FUNCTION_BLOCK TFPalletizerWorkAreaManagerTF_Lastre
VAR_INPUT
	Cfg 						: Config;
	WorkArea 					: POINTER TO ARRAY [1..MAXAREA] OF TFMachinePalletizer_WorkArea;
	WorkAreaState 				: POINTER TO ARRAY [1..MAXAREA] OF TFMachinePalletizer_WorkAreaState;
	WorkAreaOffset				: POINTER TO ARRAY [1..MAXAREA] OF TFMachinePalletizer_WorkAreaOffset;
	PX_WorkArea 				: ARRAY [1..MAXAREA] OF BOOL;
	WorkPickPoint 				: POINTER TO ARRAY [1..MAXPICKPOINT] OF TFMachinePalletizer_WorkPickPointSlab;
	WorkPickPointState 			: POINTER TO ARRAY [1..MAXPICKPOINT] OF TFMachinePalletizer_WorkPickPoint_State;
	//WorkPickPointTransportState	: POINTER TO ARRAY [1..MAXPICKPOINT] OF TFMachinePalletizer_WorkPickPointTransport_State;
	//WorkPickPointStoreState		: POINTER TO ARRAY [1..MAXPICKPOINT] OF TFMachinePalletizer_WorkPickPointStore_State;
	WorkPickPointOffset 		: POINTER TO ARRAY [1..MAXPICKPOINT] OF TFMachinePalletizer_WorkPickPointOffset;
	Forming 					: POINTER TO ARRAY [1..MAXFORMING] OF TFMachinePalletizer_FormingForSlab;
	Pallet 						: POINTER TO ARRAY [1..MAXPALLET] OF TFMachinePalletizer_Pallet;
	Layer 						: POINTER TO ARRAY [1..MAXLAYER] OF TFMachinePalletizer_Layer;
	Mission 					: POINTER TO TFMachinePalletizer_Mission;
	PickPlaceParameters			: POINTER TO TFMachinePalletizer_PickPlaceParameters;
	ExternalWaitPositionRequest : BOOL;
	ProgressiveNrWA 			: POINTER TO UDINT;
	UsedCode 					: POINTER TO ARRAY [1..MAXFORMINGCODE] OF INT;
	TCPParameter 				: POINTER TO TFModulePalletizerRobot_TCPPar;
	TilterPack 					: POINTER TO ARRAY [1..MAXHANDLINGSTACK] OF TFHandlingPack;
	PreviousPWA 				: POINTER TO UINT;
	RestoreCWA 					: POINTER TO BOOL;
	PreviousStackWA 			: POINTER TO INT;
	WorkAreaManager 			: POINTER TO TFWorkAreaManager;
	ModuleAX_X 					: POINTER TO TFModulePalletizer_Ax;
	ModuleAX_Y 					: POINTER TO TFModulePalletizer_Ax;
	ModuleAX_Z 					: POINTER TO TFModulePalletizer_Ax;
	ModuleAX_J 					: POINTER TO TFModulePalletizer_Ax;
	ModuleAX_K 					: POINTER TO TFModulePalletizer_Ax;
	
	ModulePinza					: pointer to TFModulePalletizer_Pinza;
	
	WorkAreaZone 				: POINTER TO TFMachinePalletizer_WorkAreaZone;	// Struttura delle zone di lavoro
	//HandlingPackTable : POINTER TO TFHandlingPackTable;						// Tabella contenente i pacchi sui trasporti
	ArrayPacchi 			: POINTER TO DUT_ArrayPacchi; 						//Array contenente i pacchi sui trasporti				
	GestioneAZoneAbilitata 	: POINTER TO BOOL;									// Abilitazione della gestione a zone
	HandlingRun 			: BOOL;												//Traspoti in Automatico
	RichiestaStartRibaltino : BOOL;
	AbilitaForzaturaStatoDaRiposoAPrelievo 			: POINTER TO BOOL;			// Abilita il cambio al volo della missione dal ciclo di riposo al ciclo di prelievo
	AbilitaDisposizionePalletContinua 				: POINTER TO BOOL;			// Abilitazione del deposito dei pallet ogni qualvolta il carico imposto dalla line a soddisfi determinato requisiti
	AbilitaDepositoPaccoOrrizzonataleConTasteggio 	: POINTER TO BOOL; 			// Abilitazione per il deposito del pacco con tasteggio del pacco orrizzontale
	AbilitaAssegnazioneCodicePiazzoleConPaccoSuRibaltino 	: BOOL := TRUE; 	// Abilitazione della gestione del codice in modo opportunistico rispettando le zone
	AbilitaOffsetInUscitaTasteggioPrelievoPallet 			: POINTER TO BOOL; 	// Abilitazione dell'offset in uscita dei tastatori in prelievo pallet con tasteggio
	
	//TabellaDiProduzione : POINTER TO ARRAY [1..MAXPRODLIST] OF TFMachinePalletizer_ListaProduzione; //Lista degli ordini di produzione che devo Svolgere
	
	WorkAreaProductionList : POINTER TO ARRAY [1..MAXAREA] OF TFMachinePalletizer_ListaProduzione_WAM;// ARRAY [1..MAXAREA] OF TFMachinePalletizer_ListaProduzione_WAM; //Lista di produzione che devo Svolgere PER ogni POSTAZIONE
	
	//
	RichiestaIngZonaDX : BOOL; //Richiesta di ingresso zona DX del pallettizzatore, le postazioni vanno dalla 1 alla 4
	RichiestaIngZonaSX : BOOL; //Richiesta di ingresso zona SX del pallettizzatore, le postazioni vanno dalla 5 alla 8
	
END_VAR
VAR_OUTPUT
	InWaitPosition 			: BOOL;
	DepositoPaccoInLenta 	: BOOL;					// TRUE: Il deposito del pacco deve avvenire in lenta
	ForzaPrelievoPaccoDuranteCicloDiRiposo : BOOL; 	// Indica che il ciclo sta facendo un salto: Da ciclo di riposo -> A ciclo di prelievo 
	Errore : TFError_WAM; 							//Codice di errore del WorkAreaManager
END_VAR
VAR
	i : UINT;
	TimerPositionMission : REAL;
	CurrentWorkArea : INT;
	cwa : UINT;
	pwa : UINT;
	wa : INT;
	pf : INT;
	pp : INT;
	fcode : INT;
	ppick : UINT; //Punto di prelievo
	XPick : LREAL;
	YPick : LREAL;
	ZPick : LREAL;
	JPick : LREAL;
	EnableCode : ARRAY [1..MAXFORMINGCODE*MAXFORMING] OF INT;
	WAPointer : ARRAY [1..MAXAREA] OF TFMachinePalletizer_WorkAreaSort;
	ZOffsetPick : REAL;
	ZOffsetPlace : REAL;
	WaitPositionRequest : BOOL;
	WaitPositionRequestTRIG : BOOL;
	BypassTEST 								: BOOL; // ByPASS per il conteggio dei pacchi durante le simulazioni
	CicloDiRiposoNecessario 				: BOOL;	// Forzatura del ciclo di riposo da parte del WAManager
	NPacchiPresentiSuLinea 					: UINT;	// Indica il numero dei pacchi presenti sulla linea
	NUltimiTrasportiOccupati 				: UINT;	// Indica il numero di trasporti occupati a partire dal ribaltino
	HandlingOKPrelievoPacco 				: BOOL; // Indica che il Ribaltino è pronto a consegnare il pacco
	ConsentiDepositoPaccoSuWA 				: BOOL; // Indica il Pacco può essere depositato sulla WorkArea

	DisabilitaApproccioPacciOrrizzontali 	: BOOL := TRUE; // Abilitazione dell'approccio per i pacchi orrizzontali, in questo modo il ciclo è più rapido
	QuotaFittizziaPerTasteggioDepPacchi 	: REAL := 200; 	//Quota fittizzia per consentire il tasteggio durante il deposito dei pacci orrizzontali
	UltimaPoastazioneDiAssegnazione 		: INT;	// Variabile per Debug Interno
	UltimoComando 							: INT;	// Variabile per Debug Interno
	UltimoStatoCMDRibaltino 				: INT;	// Variabile per Debug Interno
	WAconCodiceWPPPresente 					: BOOL;	// Indica che esiste almento una WA in lavorazione con il codice del pacco presente sul ribaltino in questione
	FormaturaAttivaMista 					: BOOL;	// Indica che la formatura attiva è di tipo Misto (FALSE:utilizzata per anticipare ulteriormente il ribaltino,TRUE:si aspetta che sia terminato il deposito del pacco in corso prima di comandare il ribaltino)
	PalletDepositatiSenzaCodicePresenti 	: BOOL;	// Indica che sono presenti dei pallet depositati con codice 0 ( Per assegnazione codice in modalità opportunistica(In base al codice sul ribaltino))
	CodiceValidoPerWA 						: BOOL; // Indica che il codice del pacco sul ribaltino è presente nella formatura attiva nella WA considerata

	SimulazioneSenzaPallet 					: BOOL; //Variabile per simulare in officina senza pacco e pallet
	
	FormatureMultipleAttive 				: BOOL;	//Indica che ci sono più formature Diverse ABILITATE
	////////// NUOVE PER LASTRE ////////////
	DIREZIONE_X_POSITIVA					: BOOL;
	
	TFWAM_CreaMissione_DepFaldaSuLastra 	: TFWAM_CreaMissione_DepPrelElemento;
	TFWAM_CreaMissione_DepFaldaSuPallet 	: TFWAM_CreaMissione_DepPrelElemento;
	TFWAM_CreaMissione_Destinazione			: TFWAM_CreaMissione_DepPrelElemento;
	
	TFWAM_CreaMissione_PrelLastraDaWA 		: TFWAM_CreaMissione_DepPrelElemento;
	TFWAM_CreaMissione_DepLastraDaWA		: TFWAM_CreaMissione_DepPrelElemento;
	
	TFWAM_CreaMissione_DepLastraDaPP		: TFWAM_CreaMissione_DepPrelElemento;
	
	TFWAM_CreaMissione_DepFaldaSuMagazzino 	: TFWAM_CreaMissione_DepPrelElemento;

	
	PostazioneConListaInEsecuzione : UINT; //Indica il numero della postazione avente una lista di lavorazione ion esecuzione
	WADiDepositoFinale : UINT; //WorkArea Di Desinazione della Lastra 
	NLastraDaPrelevare : INT; //Numero della lastra da prelevare = N° della prima lastra che sarà prelevata dalla cavallina
	RIESEGUI_PAREGGIATURA : BOOL; //Forzo L'esecuzione della pareggiatura della lastra Dopo arresto anomalo del ciclo
	ElList1: UINT;
	ElList : UINT;//Elemento in elaborazione nella lista
	
	
	LastRequetsID : STRING; //Ultimo ID depositato sulla rulliera dopo il depal
	LatoPrelievo : INT; //Indica il lato di prelievo per le cavalline = 90 o 180
	LastPpick : UINT; //Memoria dell'ultimo 

	debug : bool;
	ppickOld : UINT;
	ApprendimentoNulloRullieraDeposito : TFMachinePalletizer_CoordinateApprendimento;
	DisabilitaCicloRiposoPerPezzoInPresa : BOOL;
	LatoDeposito : INT; //Indica il lato di deposito.. per le cavalline = 90 o 180


	Debug_SupportoMancanteInDeposito : BOOL;//Indica che il supporto sul deposito non è presente
	Debug_RullieraInManuale : BOOL;//Indica che la rulliera è in manuale
	Debug_NessunaListaDaProcessare : BOOL;//Indica che non c'è nessuna lista da processare
	Debug_RicSupportoWA : ARRAY[1..MAXAREA] OF BOOL;//Indica una richiesta del supporto da partede della postazione
	Actual_WorkOrde: INT;
	AltezzaCentroLastraInclinata : REAL;
	AngoloPrelievo : REAL;
	QuotaLastraYRealTimePrelievo : REAL;
	QuotaLastraYRealTimeDeposito : REAL;
	QuotaLastraZRealTimePrelievo : REAL;
	QuotaLastraZRealTimeDeposito : REAL;
	
	TFCalcoloFormaturaDaLista	: Calcolo_Formatura_Completa;//FB per il calcolo della formatura
	CalcolaFormaturaTrig : BOOL;
	
	PplaceOld : UINT;
	AngoloDepositoLastra : REAL;
	
	Y_PuntoPrelievo0: REAL;
	Y_PuntoPrelievo180: REAL;
	OffSetY180Cavallete: REAL;
	AguloDeRecogida: UINT;
	AguloDeDeposito: UINT;
END_VAR

(* Set variabili varie *)
Errore.Code:= 0;
Errore.Extracode:=0;

(* Chiamata del timer per andare alla posizione di riposo *)
TFTimerCall(ADR(TimerPositionMission),Cfg.TimeBase);
(* Inizializzazione del WAM *)
IF WorkAreaManager^.State = -1 THEN
	WorkAreaManager^.State := WAMANAGER_NOP;
	ExternalWaitPositionRequest := TRUE;
END_IF

EnableCode := TFGetEnableCode_Lastre(Forming);



IF Mission^.State <> MISSION_STATE_NOP THEN
	TFTimerSet(ADR(TimerPositionMission),300,TRUE);
END_IF
IF ((ExternalWaitPositionRequest AND WorkAreaManager^.State = WAMANAGER_NOP)  OR TFTimerDone(ADR(TimerPositionMission))) AND NOT InWaitPosition THEN
	CicloDiRiposoNecessario	:= TRUE;
	WaitPositionRequestTRIG := TRUE;
END_IF
IF 	WaitPositionRequestTRIG THEN
	WaitPositionRequest := TRUE;
END_IF
IF WaitPositionRequestTRIG AND WaitPositionRequest AND (InWaitPosition AND WorkAreaManager^.State = WAMANAGER_NOP) THEN
	WaitPositionRequest := FALSE;
	WaitPositionRequestTRIG := FALSE;
END_IF


CASE WorkAreaManager^.State OF
	WAMANAGER_NOP:
			
		IF RichiestaIngZonaSX THEN
			Mission^.PPick			:= 5;
			Mission^.TPick 			:= TPICK_NOT_DEFINED;
			Mission^.XPick			:= WorkArea^[5].X;
			Mission^.YPick			:= WorkSpace.Y/2 + OffSetPosYReposo;//Workarea^[5].Y;
			Mission^.ZPick			:= ModuleAX_Z^.Ax^.Parameter.MAXPosition - 100 -OffsetSicurezza.Z.Avuoto; // estaba 100
			
			Mission^.JPick			:= 90;
			
			Mission^.PPlace			:= Mission^.PPick;
			Mission^.XPlace			:= Mission^.XPick;
			Mission^.YPlace			:= Mission^.YPick;
			Mission^.ZPlace			:= Mission^.ZPick;
			Mission^.JPlace			:= Mission^.JPick;

			Mission^.XDim 	:= 0;
			Mission^.YDim	:= 0;
			Mission^.ZDim	:= 0;
			
			X_Riposo := Mission^.XPick;
			Y_Riposo := Mission^.YPick;
			Z_Riposo := Mission^.ZPick;
			J_Riposo := Mission^.JPick;
			
			(* Set della condizione di posizione di riposo Wait Position *)
			InWaitPosition := TFPalletizerInPosizioneRiposo(ModuleAX_X,ModuleAX_Y,ModuleAX_Z,ModuleAX_J,Mission);

			IF WaitPositionRequest AND NOT InWaitPosition AND
			(ExternalWaitPositionRequest OR CicloDiRiposoNecessario) THEN //Se la macchina non è a riposo, ce la mando
				WorkAreaManager^.State := WAMANAGER_CICLO_RIPOSO_INIT;
			ELSE	//Se la macchina è ferma e a riposo -> verifica eventuali cambi di produzione
				ReadyToChange := TRUE;
			END_IF

		ELSIF RichiestaIngZonaDX THEN
			Mission^.PPick			:= 1;
			Mission^.TPick 			:= TPICK_NOT_DEFINED;
			Mission^.XPick			:= WorkArea^[4].X;
			Mission^.YPick			:= WorkSpace.Y/2 + OffSetPosYReposo;//Workarea^[1].Y;
			Mission^.ZPick			:= ModuleAX_Z^.Ax^.Parameter.MAXPosition - 100 -OffsetSicurezza.Z.Avuoto ;
			Mission^.JPick			:= 90;
			
			Mission^.PPlace			:= Mission^.PPick;
			Mission^.XPlace			:= Mission^.XPick;
			Mission^.YPlace			:= Mission^.YPick;
			Mission^.ZPlace			:= Mission^.ZPick;
			Mission^.JPlace			:= Mission^.JPick;

			Mission^.XDim 	:= 0;
			Mission^.YDim	:= 0;
			Mission^.ZDim	:= 0;
			
			X_Riposo := Mission^.XPick;
			Y_Riposo := Mission^.YPick;
			Z_Riposo := Mission^.ZPick;
			J_Riposo := Mission^.JPick;

			(* Set della condizione di posizione di riposo Wait Position *)
			InWaitPosition := TFPalletizerInPosizioneRiposo(ModuleAX_X,ModuleAX_Y,ModuleAX_Z,ModuleAX_J,Mission);
			
			IF WaitPositionRequest AND NOT InWaitPosition AND
			(ExternalWaitPositionRequest OR CicloDiRiposoNecessario) THEN //Se la macchina non è a riposo, ce la mando
				WorkAreaManager^.State := WAMANAGER_CICLO_RIPOSO_INIT;
			ELSE	//Se la macchina è ferma e a riposo -> verifica eventuali cambi di produzione
				ReadyToChange := TRUE;
			END_IF
		ELSE
		 	Mission^.PPick			:= 1;
			Mission^.TPick 			:= TPICK_NOT_DEFINED;
			Mission^.XPick			:= ModuleAX_X^.Ax^.Status.ActPosition;// WorkArea^[1].X;
			Mission^.YPick			:= WorkSpace.Y/2 + OffSetPosYReposo;//Workarea^[1].Y;
			Mission^.ZPick			:= ModuleAX_Z^.Ax^.Parameter.MAXPosition - 100 - OffsetSicurezza.Z.Avuoto; 
			Mission^.JPick			:= 90;
			
			Mission^.PPlace			:= Mission^.PPick;
			Mission^.XPlace			:= Mission^.XPick;
			Mission^.YPlace			:= Mission^.YPick;
			Mission^.ZPlace			:= Mission^.ZPick;
			Mission^.JPlace			:= Mission^.JPick;

			Mission^.XDim 	:= 0;
			Mission^.YDim	:= 0;
			Mission^.ZDim	:= 0;
			
			X_Riposo := Mission^.XPick;
			Y_Riposo := Mission^.YPick;
			Z_Riposo := Mission^.ZPick;
			J_Riposo := Mission^.JPick;

			(* Set della condizione di posizione di riposo Wait Position *)
			InWaitPosition := TFPalletizerInPosizioneRiposo(ModuleAX_X,ModuleAX_Y,ModuleAX_Z,ModuleAX_J,Mission);
			
			IF WaitPositionRequest AND NOT InWaitPosition AND
			(ExternalWaitPositionRequest OR CicloDiRiposoNecessario) THEN //Se la macchina non è a riposo, ce la mando
				WorkAreaManager^.State := WAMANAGER_CICLO_RIPOSO_INIT;
			ELSE	//Se la macchina è ferma e a riposo -> verifica eventuali cambi di produzione
				ReadyToChange := TRUE;
			END_IF
		END_IF
						
	WAMANAGER_CICLO_RIPOSO_INIT:
	 	
		IF RichiestaIngZonaSX THEN
			Mission^.PPick			:= 5;
			Mission^.TPick 			:= TPICK_NOT_DEFINED;
			IF AreaPikingConCavallete AND MultiplesCavalletesReceta OR WorkAreaState^[PosRobot].Supporto.Tipologia = CAVALLETTO 
				OR (PosRobot <> 0 AND  HMI_WorkAreaDataPicking[PosRobot].Typology = CAVALLETTO)	THEN
				Mission^.XPick			:= WorkArea^[PosFinOrdenPikingCaballete].X;
				Mission^.YPick			:= ModuleAX_y^.Ax^.AxRef^.NcToPlc.ActPos;
				Mission^.ZPick			:= ModuleAX_Z^.Ax^.Parameter.MAXPosition - 100 -OffsetSicurezza.Z.Avuoto;
				Mission^.JPick			:= ModuleAX_j^.Ax^.AxRef^.NcToPlc.ActPos ;
			ELSE
				Mission^.XPick			:= WorkArea^[5].X;
				Mission^.YPick			:= WorkSpace.Y/2 + OffSetPosYReposo;//Workarea^[5].Y;
				Mission^.ZPick			:= ModuleAX_Z^.Ax^.Parameter.MAXPosition - 100 -OffsetSicurezza.Z.Avuoto;
				Mission^.JPick			:= 90;
			END_IF
			
			Mission^.PPlace			:= Mission^.PPick;
			Mission^.XPlace			:= Mission^.XPick;
			Mission^.YPlace			:= Mission^.YPick;
			Mission^.ZPlace			:= Mission^.ZPick;
			Mission^.JPlace			:= Mission^.JPick;

			Mission^.XDim 	:= 0;
			Mission^.YDim	:= 0;
			Mission^.ZDim	:= 0;
			
			X_Riposo := Mission^.XPick;
			Y_Riposo := Mission^.YPick;
			Z_Riposo := Mission^.ZPick;
			J_Riposo := Mission^.JPick;

		ELSIF RichiestaIngZonaDX THEN
			Mission^.PPick			:= 1;
			Mission^.TPick 			:= TPICK_NOT_DEFINED;
			IF AreaPikingConCavallete AND MultiplesCavalletesReceta OR WorkAreaState^[PosRobot].Supporto.Tipologia = CAVALLETTO 
				OR (PosRobot <> 0 AND  HMI_WorkAreaDataPicking[PosRobot].Typology = CAVALLETTO) THEN
				Mission^.XPick			:= WorkArea^[PosFinOrdenPikingCaballete].X;
				Mission^.YPick			:= ModuleAX_y^.Ax^.AxRef^.NcToPlc.ActPos;
				Mission^.ZPick			:= ModuleAX_Z^.Ax^.Parameter.MAXPosition - 100 -OffsetSicurezza.Z.Avuoto;
				Mission^.JPick			:= ModuleAX_j^.Ax^.AxRef^.NcToPlc.ActPos ;
				
				
			ELSE
				Mission^.XPick			:= WorkArea^[4].X;
				Mission^.YPick			:= WorkSpace.Y/2+OffSetPosYReposo;//Workarea^[1].Y;
				Mission^.ZPick			:= ModuleAX_Z^.Ax^.Parameter.MAXPosition - 100 -OffsetSicurezza.Z.Avuoto;
				Mission^.JPick			:= 90;
			END_IF
			
			
			Mission^.PPlace			:= Mission^.PPick;
			Mission^.XPlace			:= Mission^.XPick;
			Mission^.YPlace			:= Mission^.YPick;
			Mission^.ZPlace			:= Mission^.ZPick;
			Mission^.JPlace			:= Mission^.JPick;

			Mission^.XDim 	:= 0;
			Mission^.YDim	:= 0;
			Mission^.ZDim	:= 0;
			
			X_Riposo := Mission^.XPick;
			Y_Riposo := Mission^.YPick;
			Z_Riposo := Mission^.ZPick;
			J_Riposo := Mission^.JPick;
		ELSE
		 	Mission^.PPick			:= 1;
			Mission^.TPick 			:= TPICK_NOT_DEFINED;
			IF AreaPikingConCavallete AND MultiplesCavalletesReceta OR WorkAreaState^[PosRobot].Supporto.Tipologia = CAVALLETTO
				OR (PosRobot <> 0 AND  HMI_WorkAreaDataPicking[PosRobot].Typology = CAVALLETTO) THEN
				Mission^.XPick			:= WorkArea^[PosFinOrdenPikingCaballete].X;
				Mission^.YPick			:= ModuleAX_y^.Ax^.AxRef^.NcToPlc.ActPos;
				Mission^.ZPick			:= ModuleAX_Z^.Ax^.Parameter.MAXPosition - 100 -OffsetSicurezza.Z.Avuoto;
				Mission^.JPick			:= ModuleAX_j^.Ax^.AxRef^.NcToPlc.ActPos ;
			ELSE
				Mission^.XPick			:= ModuleAX_X^.Ax^.Status.ActPosition;// WorkArea^[1].X;
				Mission^.YPick			:= (*2000   *)   WorkSpace.Y/2+OffSetPosYReposo;//Workarea^[1].Y ;
				Mission^.ZPick			:= ModuleAX_Z^.Ax^.Parameter.MAXPosition - 100 - OffsetSicurezza.Z.Avuoto;
				Mission^.JPick			:= 90;
			END_IF
			
			
			Mission^.PPlace			:= Mission^.PPick;
			Mission^.XPlace			:= Mission^.XPick;
			Mission^.YPlace			:= Mission^.YPick;
			Mission^.ZPlace			:= Mission^.ZPick;
			Mission^.JPlace			:= Mission^.JPick;

			Mission^.XDim 	:= 0;
			Mission^.YDim	:= 0;
			Mission^.ZDim	:= 0;
			
			X_Riposo := Mission^.XPick;
			Y_Riposo := Mission^.YPick;
			Z_Riposo := Mission^.ZPick;
			J_Riposo := Mission^.JPick;
		END_IF
	WorkAreaManager^.State  := WAMANAGER_CICLO_RIPOSO_RUN;
		
	WAMANAGER_CICLO_RIPOSO_RUN:
		
		IF Mission^.State = MISSION_STATE_VAIaRIPOSO_RUN THEN
			;
		ELSIF Mission^.State = MISSION_STATE_VAIaRIPOSO_END THEN
			CicloDiRiposoNecessario := FALSE;
			WorkAreaManager^.State 	:= WAMANAGER_CICLO_RIPOSO_END;	// setto lo stato del WAMANAGER
		ELSIF Mission^.State = MISSION_STATE_ERROR THEN
			;
		END_IF
		
	WAMANAGER_CICLO_RIPOSO_END:
		WorkAreaManager^.State := WAMANAGER_NOP;
		
	WAMANAGER_SALTA_DA_RIPOSO_A_PRELIEVO:
		IF Mission^.State = MISSION_STATE_VAIaRIPOSO_END THEN
			WorkAreaManager^.State 	:= WAMANAGER_NOP;	// setto lo stato del WAMANAGER
		END_IF
	ELSE;					
END_CASE


(*Con Stop in Fase, solo se la Missione è NOP vado in WAIT *)
IF NOT WaitPositionRequest OR 
	(WaitPositionRequest AND WorkAreaManager^.State <> WAMANAGER_NOP AND WorkAreaManager^.State <> WAMANAGER_CICLO_RIPOSO_RUN  AND WorkAreaManager^.State <> WAMANAGER_CICLO_RIPOSO_INIT) THEN
	WAPointer := TFGetNearestWA(WorkArea,WorkPickPoint^[PICKPOINT1]);
	FOR pwa:=1 TO MAXAREAPRESENT DO	
		pwa := RestoringCWA(RestoreCWA,PreviousPWA,pwa);
		RestoreCWA^ := FALSE;		
		cwa := WAPointer[pwa].cwa;
		cwa := pwa;
		IF PreviousStackWA^ < 0 THEN
			PreviousStackWA^ := 1;
		END_IF
		
		(* Ciclo solo nelle postazioni in cui non è attiva la richiesta di ingresso.. in questo modo la macchina non cercherà di lavorare dove c'è l'operatore *)
		IF RichiestaIngZonaSX THEN
			IF cwa > 4 THEN
				CONTINUE;
			END_IF
		ELSIF RichiestaIngZonaDX THEN
			IF cwa < 5 THEN
				CONTINUE;
			END_IF
		ELSE
		 	;
		END_IF
		
		CASE WorkAreaState^[cwa].State OF	
(**********************************************************************************************************************************************************************************)
(**********************************************************************************************************************************************************************************)
		(* POSTAZIONE LIBERA E ABILITATA *)
(**********************************************************************************************************************************************************************************)
(**********************************************************************************************************************************************************************************)
			WORKAREA_STATE_FREE_ENABLED:

				CASE TIPOLOGIA_FUNZIONAMENTO_MACCHINA OF 
					
					FUNZIONAMENTO_SLAVE:;{info "Implementare logica utilizzata WAM nel magazzino lastre di ariostea!!!"}
			
					FUNZIONAMENTO_PICKING:
						{Region "TIPOLOGIA POSTAZIONE"}
							(* Se la postazione è ABILITATA *)			
							IF WorkArea^[cwa].Enable = 1 THEN
								(* Se la FTC di presenza è SPENTA *)
								//IF NOT PX_WorkArea[cwa] THEN
									(* Valuto la tipologia di postazione *)
									CASE WorkArea^[cwa].Typology OF
										(* Per Postazione Di Lavoro INDEFINITE *)	
										TYPOLOGY_NOT_DEFINED:
											CONTINUE;//Passo alla postazione successiva nel ciclo FOR							
										(* Per Postazione di Lavoro *)
										TYPOLOGY_PALLET:
											 	WorkAreaState^[cwa].P := -1;
												IF cwa <> NumPostazioneSuRulliera THEN
													IF PX_WorkArea[cwa] THEN // Con presenza vado in lavorazione altrimenti forzo chiamata LGV
														WorkAreaState^[cwa].State := WORKAREA_STATE_OCCUPIED_WORKING;
													ELSE
														//WorkAreaState^[cwa].LGV_Req 			:= REQ_LGV; //Setto la chiamata
														//WorkAreaState^[cwa].LGV_GetIn_GetOut 	:= REQ_DEPOSITO_LGV_VUOTO;//Setto la tipologia di chiamata
														;//WorkAreaState^[cwa].State 				:= WORKAREA_STATE_FREE_LGVREQ;
													END_IF
												END_IF
										(* Per Magazzino di Lavoro di tipo Falde *)
										TYPOLOGY_LAYER:							
											CASE WorkArea^[cwa].Typology_Desc OF
												(* WorkArea di tipo *) 
												MAGAZZINO_FALDE_IN_WA: 	
													WorkAreaState^[cwa].Taped := -1;
													WorkAreaState^[cwa].P := -1;
													IF PX_WorkArea[cwa] THEN // Con presenza vado in lavorazione altrimenti forzo chiamata LGV
														WorkAreaState^[cwa].State := WORKAREA_STATE_OCCUPIED_WORKING;
													ELSE
														WorkAreaState^[cwa].State := WORKAREA_STATE_FREE_LGVREQ;
													END_IF	
												
												(* PickPoint di tipo *)
												MAGAZZINO_FALDE_IN_PP:	
													WorkAreaState^[cwa].Taped := -1;
													WorkAreaState^[cwa].P := -1;
													IF PX_WorkArea[cwa] THEN // Con presenza vado in lavorazione altrimenti forzo chiamata LGV
														WorkAreaState^[cwa].State := WORKAREA_STATE_OCCUPIED_WORKING;
													ELSE
														WorkAreaState^[cwa].State := WORKAREA_STATE_FREE_ENABLED;
													END_IF	
											END_CASE
												
										(* Tipologia Postazione ESTERNA al perimetro del Pallettizzatore: 
										Utilizzata per deposito o prelievo di Pallet/Casse/Cavalline lavorate o da lavorare *)	
										TYPOLOGY_EXTERNAL_DEPPREL:;
										TYPOLOGY_OVER_TRANSPORT:
											Debug_RicSupportoWA[cwa] := FALSE;
											IF WorkAreaState^[cwa].TransportState.ProdPresence = WORKPICKPOINT_PRODOTTO_PRESENTE THEN // Con presenza vado in lavorazione altrimenti sto in attesa che sia presente qualcosa
												WorkAreaState^[cwa].State := WORKAREA_STATE_OCCUPIED_WORKING;
											ELSIF WorkAreaState^[cwa].TransportState.ProdPresence <> WORKPICKPOINT_PRODOTTO_PRESENTE AND cwa = NumPostazioneSuRulliera THEN
												(* Ricavo se una postazione ha una Lista in esecuzione *)
												PostazioneConListaInEsecuzione := TFWAM_RicavaListaInLavoro(WorkAreaProductionList := WorkAreaProductionList);
												(* Se non ho liste in esecuzione e ho una lista da eseguire sulla postazione, vado a richiedere il suporto *)
												IF (WorkAreaProductionList^[cwa].Stato = LISTA_PROD_DA_ESEGUIRE AND PostazioneConListaInEsecuzione = 0) THEN 
													Debug_RicSupportoWA[cwa] := TRUE;
												END_IF			
												WorkAreaState^[cwa].State := WORKAREA_STATE_FREE_ENABLED;
											END_IF	
										TYPOLOGY_BUNDLE:
											IF WorkAreaState^[cwa].TransportState.ProdPresence = WORKPICKPOINT_PRODOTTO_PRESENTE THEN // Con presenza vado in lavorazione altrimenti sto in attesa che sia presente qualcosa
												WorkAreaState^[cwa].State := WORKAREA_STATE_OCCUPIED_WORKING;
											ELSE
												WorkAreaState^[cwa].State := WORKAREA_STATE_FREE_ENABLED;
											END_IF
									ELSE
										CONTINUE;//Passo alla postazione successiva nel ciclo FOR	
									END_CASE	
								(* Se la FTC di presenza è ACCESA *)	
								//ELSE
									(* Genero Errore relativo a FTC oscurata senza la presenza LOGICA*)
									//Errore.Code 	 := ErrWAM_FTCWA_ON_PrenzaLogicaOFF;
									//Errore.ExtraCode := cwa;
								//END_IF
							(* Se la postazione è DISABILITATA *)	
							ELSIF WorkArea^[cwa].Enable < 1 THEN
								IF PX_WorkArea[cwa] THEN (* CON FTC di presenza Assegno stato in Occupata e Disabilitata *)
									WorkAreaState^[cwa].State := WORKAREA_STATE_OCCUPIED_DISABLED;
								ELSE					(* SENZA FTC di presenza Asegno stato in LIBERA e Disabilitata *)
									WorkAreaState^[cwa].State := WORKAREA_STATE_FREE_DISABLED;
								END_IF
							END_IF
						{endregion}

				ELSE //riferito a TIPOLOGIA_FUNZIONAMENTO_MACCHINA
				;
				END_CASE

(**********************************************************************************************************************************************************************************)
(**********************************************************************************************************************************************************************************)			
			(* Free Disabled *)
(**********************************************************************************************************************************************************************************)
(**********************************************************************************************************************************************************************************)
			WORKAREA_STATE_FREE_DISABLED:
				(* Se la postazione è ABILITATA *)
				IF WorkArea^[cwa].Enable = 1 THEN
					(* Se la FTC di presenza è SPENTA *)
					//IF NOT PX_WorkArea[cwa] THEN
						WorkAreaState^[cwa].State := WORKAREA_STATE_FREE_ENABLED;
					(* Se la FTC di presenza è ACCESA *)
					//ELSE
						(* Genero Errore relativo a FTC oscurata senza la presenza LOGICA*)
						//Errore.Code 	 := ErrWAM_FTCWA_ON_PrenzaLogicaOFF;
						//Errore.ExtraCode := cwa;
						//IF CWA = NumPostazioneFALDE THEN
						//	Errore.Code := ErrMODULEPALLETIZERROBOT_EMPTYLAYERSTACK;
						//END_IF
					//END_IF	
				(* Se la postazione è DISABILITATA *)
				ELSIF WorkArea^[cwa].Enable < 1 THEN
					IF PX_WorkArea[cwa] THEN (* CON FTC di presenza Assegno stato in Occupata e Disabilitata *)
						WorkAreaState^[cwa].State := WORKAREA_STATE_OCCUPIED_DISABLED;
					ELSE					(* SENZA FTC di presenza Asegno stato in LIBERA e Disabilitata *)
						WorkAreaState^[cwa].State := WORKAREA_STATE_FREE_DISABLED;
					END_IF	
				END_IF
(**********************************************************************************************************************************************************************************)
(**********************************************************************************************************************************************************************************)
			(* Occupied + Disabled *)
(**********************************************************************************************************************************************************************************)
(**********************************************************************************************************************************************************************************)
			WORKAREA_STATE_OCCUPIED_DISABLED:
				(* Nessuna Operazione! Si PROSEGUE LA LAVORAZIONE se viene Abilitata la Piazzola *)
				(* Se la postazione è ABILITATA e la Formatura è ABILITATA *)
				IF WorkArea^[cwa].Enable = 1  AND  (Forming^[WorkAreaState^[cwa].F].Enable = 1 OR PX_WorkArea[cwa]) THEN
					WorkAreaState^[cwa].State := WORKAREA_STATE_OCCUPIED_WORKING;
				END_IF
(**********************************************************************************************************************************************************************************)
(**********************************************************************************************************************************************************************************)	
			(* Free + Working (Gestione PALLET VUOTO) *)
(**********************************************************************************************************************************************************************************)
(**********************************************************************************************************************************************************************************)
			WORKAREA_STATE_FREE_WORKING:
				IF PreviousStackWA^ < 0 THEN
					PreviousStackWA^ := 1;
				END_IF
				(* Se la postazione è ABILITATA *)			
				IF WorkArea^[cwa].Enable = 1 THEN
					(* Se la FTC di presenza è SPENTA *)
					IF NOT PX_WorkArea[cwa] THEN
						CASE WorkAreaManager^.State OF
							WAMANAGER_NOP:;
							
						ELSE		(* riferito al case WorkAreaManager^.State *)
							;
						END_CASE	(* riferito al case WorkAreaManager^.State *)
					(* Se la FTC di presenza è ACCESA *)
					ELSE
						WorkAreaState^[cwa].State := WORKAREA_STATE_OCCUPIED_WORKING;
						(* Genero Errore relativo a Ftocellula oscurata senza la presenza LOGICA*)
						//Errore.Code 	 := ErrWAM_FTCWA_ON_PrenzaLogicaOFF;
						//Errore.ExtraCode := cwa;
					END_IF
				
				(* Se la postazione è DISABILITATA *)
				ELSIF WorkArea^[cwa].Enable < 1 THEN
					(* Controllo della Ph di presenza pallet, in base a quello gestisco lo stato della piazzola *)
					IF PX_WorkArea[cwa] THEN
						WorkAreaState^[cwa].State := WORKAREA_STATE_OCCUPIED_DISABLED;
					ELSE
						WorkAreaState^[cwa].State := WORKAREA_STATE_FREE_DISABLED;
					END_IF
				END_IF
(**********************************************************************************************************************************************************************************)
(**********************************************************************************************************************************************************************************)
			(* Occupied + Working (Gestione LASTRE/FALDE) *)
(**********************************************************************************************************************************************************************************)
(**********************************************************************************************************************************************************************************)
			WORKAREA_STATE_OCCUPIED_WORKING:
				IF (WorkArea^[cwa].Enable = 1 AND ((Forming^[WorkAreaState^[cwa].F].Enable = 1 AND TIPOLOGIA_FUNZIONAMENTO_MACCHINA <> FUNZIONAMENTO_DEPAL) OR TIPOLOGIA_FUNZIONAMENTO_MACCHINA = FUNZIONAMENTO_PICKING))  OR
					((WorkArea^[cwa].Enable = 0 OR Forming^[WorkAreaState^[cwa].F].Enable = 0) AND Mission^.State > MISSION_STATE_NOP)THEN //AND
					//WorkAreaProductionList^[cwa].Stato <> LISTA_PROD_ASSENTE AND WorkAreaProductionList^[cwa].Stato <> LISTA_PROD_ESEGUITA THEN
					IF WorkAreaState^[cwa].P = 0 THEN
						WorkAreaState^[cwa].P := 1;
					END_IF
					
					CASE WorkAreaManager^.State OF							
						WAMANAGER_NOP:							
							CASE TIPOLOGIA_FUNZIONAMENTO_MACCHINA OF 
								FUNZIONAMENTO_SLAVE:;
								
								FUNZIONAMENTO_PICKING:
									Debug_SupportoMancanteInDeposito := FALSE;
									Debug_RullieraInManuale := FALSE;
									Debug_NessunaListaDaProcessare:=FALSE;
									
									(* Forzatura espulsione da HMI *)
									IF HMI_COMMAND_PAL.HMI_ForzaEspulsioneWA[cwa] THEN
										WorkAreaState^[cwa].State := WORKAREA_STATE_OCCUPIED_WORKED;
										//HMI_COMMAND_PAL.HMI_ForzaEspulsioneWA[cwa] := FALSE;
										CONTINUE;
									END_IF	
									(* Ricavo se una postazione ha una Lista in esecuzione *)
									PostazioneConListaInEsecuzione := TFWAM_RicavaListaInLavoro(WorkAreaProductionList := WorkAreaProductionList);
									
									IF WorkAreaProductionList^[cwa].Stato = LISTA_PROD_DA_ESEGUIRE AND PostazioneConListaInEsecuzione = 0 THEN
										WorkAreaProductionList^[cwa].Stato := LISTA_PROD_IN_ESECUZIONE;
										ActualPickingListFromHMI[WorkAreaProductionList^[cwa].NumeroListaAssociata].State := e_StatoWorkOrder.IN_ESECUZIONE;
									END_IF
									
									PostazioneConListaInEsecuzione := TFWAM_RicavaListaInLavoro(WorkAreaProductionList := WorkAreaProductionList);
																		
									IF (WorkAreaProductionList^[cwa].Stato = LISTA_PROD_DA_ESEGUIRE AND PostazioneConListaInEsecuzione = 0) OR 
										(WorkAreaProductionList^[cwa].Stato = LISTA_PROD_IN_ESECUZIONE AND PostazioneConListaInEsecuzione = cwa) THEN
										FOR ElList := 1 TO MAXELEMENTLIST DO
											IF WorkAreaProductionList^[cwa].NumeroListaAssociata > 0 AND_THEN 
												ElList > ActualPickingListFromHMI[WorkAreaProductionList^[cwa].NumeroListaAssociata].SlabNumber THEN
													WorkAreaProductionList^[cwa].Stato := LISTA_PROD_ESEGUITA;
													ActualPickingListFromHMI[WorkAreaProductionList^[cwa].NumeroListaAssociata].State := e_StatoWorkOrder.TERMINATO;
													EXIT;
											ELSIF WorkAreaProductionList^[cwa].PElementList[ElList].Stato = ELEMENTO_DA_ELABORARE THEN //Se l'elemento è da elaborare
												IF WorkAreaProductionList^[cwa].PElementList[ElList].WA_DEPOSITO = cwa THEN 	//Se la postazione di deposito è quella che sto considerando,Proseguo con la creazione della missione
													//IF Forming^[WorkAreaState^[cwa].F].PElement[WorkAreaState^[cwa].P].Typology = LASTRA OR  //Controllo x sicurezza che la Formatura della Postazione Chiami una Lastra o 
													//Forming^[WorkAreaState^[cwa].F].PElement[WorkAreaState^[cwa].P].Typology = FALDA THEN //Una Falda
													
													CASE WorkArea^[cwa].Typology OF
															TYPOLOGY_PALLET:	(* Tipologia Postazione Di Lavoro in WorkArea *)
																	(* Verifico che ci sia il supporto *)
																	IF PX_WorkArea[cwa] THEN
																		(* Verifico che il supporto sulla postazione di deposito coincida con il supporto previsto dalla lista di produzione *)
																		IF WorkAreaProductionList^[cwa].Support.Tipologia = WorkAreaState^[cwa].Supporto.Tipologia AND
																			(WorkAreaProductionList^[cwa].Support.XDim = WorkAreaState^[cwa].Supporto.XDim) AND
																			(WorkAreaProductionList^[cwa].Support.YDim = WorkAreaState^[cwa].Supporto.YDim) AND
																			(WorkAreaProductionList^[cwa].Support.ZDim = WorkAreaState^[cwa].Supporto.ZDim) THEN
																			CASE WorkAreaProductionList^[cwa].PElementList[ElList].PElement.Typology OF //(*WorkAreaState^[cwa].P*).PElement.Typology OF
																				LASTRA:
																						IF PX_WorkArea[WorkAreaProductionList^[cwa].PElementList[ElList].WA_PRELIEVO] THEN
																							IF WorkAreaState^[WorkAreaProductionList^[cwa].PElementList[ElList].WA_PRELIEVO].P > 1 THEN
																								WorkAreaManager^.State  := WAMANAGER_CICLO_LASTRA_WA_INIT;	(* Setto lo stato del WAMANAGER *)
																								WADiDepositoFinale := cwa; //Memorizzo la Postazione FINALE di deposito
																								Mission^.PPick	:= WorkAreaProductionList^[cwa].PElementList[ElList].WA_PRELIEVO; (* valorizzo il punto di prelievo *)
																								RestoreCWA^ := TRUE;
																								PreviousPWA^ := pwa;
																								EXIT;
																							ELSE
																								Errore.Code := ErrWA_NumPezzInPrelErrato;
																								EXIT;
																							END_IF
																						ELSE
																							Errore.Code := ErrWAM_FTCWA_OFF_PrenzaLogicaON;
																							EXIT;
																						END_IF
																				FALDA:											
																						WorkAreaManager^.State  := WAMANAGER_CICLO_FALDA_INIT;	(* Setto lo stato del WAMANAGER *)
																						WADiDepositoFinale := cwa; //Memorizzo la Postazione FINALE di deposito
																						RestoreCWA^ := TRUE;
																						PreviousPWA^ := pwa;
																						EXIT;
																				TERMINATORE:
																						WorkAreaProductionList^[cwa].Stato := LISTA_PROD_ESEGUITA;
																						RestoreCWA^ := TRUE;
																						PreviousPWA^ := pwa;
																						EXIT;																
																				
																			END_CASE
																		ELSE
																			Errore.Code := ErrWA_SupportoInDepositoErrato;//Genero l'errore che mi indica che il supporto in lavoro non coincide col supporto richiesto
																			WorkAreaManager^.State 	:= WAMANAGER_NOP;	// setto lo stato del WAMANAGER
																			EXIT;
																		END_IF
																	ELSE
																		WorkAreaManager^.State 	:= WAMANAGER_NOP; // setto lo stato del WAMANAGER
																		Debug_SupportoMancanteInDeposito := TRUE; 
																		EXIT;
																	END_IF
																
															TYPOLOGY_OVER_TRANSPORT:   (* Tipologia Di Postazione di prelievo/deposito su trasporti (rulliere o catenaria) *)
																(* Verifico che la linea sia in automatico *)		
																IF WorkAreaState^[cwa].TransportState.State = WORKPICKPOINT_STATE_AUTO THEN
																	(* Verifico che ci sia il supporto *)
																	IF WorkAreaState^[cwa].TransportState.ProdPresence = WORKPICKPOINT_PRODOTTO_PRESENTE THEN
																		(* Verifico che il supporto sulla postazione di deposito coincida con il supporto previsto dalla lista di produzione *)
																		IF WorkAreaProductionList^[cwa].Support.Tipologia = WorkAreaState^[cwa].Supporto.Tipologia AND
																			(WorkAreaProductionList^[cwa].Support.XDim = WorkAreaProductionList^[cwa].Support.XDim) AND
																			(WorkAreaProductionList^[cwa].Support.YDim = WorkAreaProductionList^[cwa].Support.YDim) AND
																			(WorkAreaProductionList^[cwa].Support.ZDim = WorkAreaProductionList^[cwa].Support.ZDim) THEN
																			CASE WorkAreaProductionList^[cwa].PElementList[WorkAreaState^[cwa].P].PElement.Typology OF
																				LASTRA:
																						WorkAreaManager^.State  := WAMANAGER_CICLO_LASTRA_WA_INIT;	(* Setto lo stato del WAMANAGER *)
																						WADiDepositoFinale := cwa; //Memorizzo la Postazione FINALE di deposito
																						RestoreCWA^ := TRUE;
																						PreviousPWA^ := pwa;
																						EXIT;
																				FALDA:											
																						WorkAreaManager^.State  := WAMANAGER_CICLO_FALDA_INIT;	(* Setto lo stato del WAMANAGER *)
																						WADiDepositoFinale := cwa; //Memorizzo la Postazione FINALE di deposito
																						RestoreCWA^ := TRUE;
																						PreviousPWA^ := pwa;
																						EXIT;
																				TERMINATORE:
																						WorkAreaProductionList^[cwa].Stato := LISTA_PROD_ESEGUITA;
																						RestoreCWA^ := TRUE;
																						PreviousPWA^ := pwa;
																						EXIT;																
																				
																			END_CASE
																		ELSE
																			Errore.Code := ErrWA_SupportoInDepositoErrato;//Genero l'errore che mi indica che il supporto in lavoro non coincide col supporto richiesto
																			WorkAreaManager^.State 	:= WAMANAGER_NOP;	// setto lo stato del WAMANAGER
																			EXIT;
																		END_IF
																	ELSE
																		WorkAreaManager^.State 	:= WAMANAGER_NOP; // setto lo stato del WAMANAGER
																		Debug_SupportoMancanteInDeposito := TRUE; 
																		EXIT;
																	END_IF
																ELSE
																	WorkAreaManager^.State 	:= WAMANAGER_NOP; // setto lo stato del WAMANAGER
																	Debug_RullieraInManuale := TRUE;
																	EXIT;
																END_IF
															
															TYPOLOGY_BUNDLE:;  (* Tipologia Di Postazione Di deposito = BUNDLE *)
															TYPOLOGY_ALIGNER:;   (* Tipologia Di Postazione Di PAREGGIATURA *)
															TYPOLOGY_EXTERNAL_DEPPREL:;(* Tipologia Postazione ESTERNA al perimetro del Pallettizzatore: Utilizzata per deposito o prelievo di Pallet/Casse/Cavalline lavorate o da lavorare *)

													END_CASE
													
													//ELSIF Forming^[WorkAreaState^[cwa].F].PElement[WorkAreaState^[cwa].P].Typology = TERMINATORE THEN //Se ho depostitato tutti gli elementi e la deposizione è completa, la evacuo	
													//	WorkAreaState^[cwa].State := WORKAREA_STATE_OCCUPIED_WORKED;
													//END_IF
												ELSE //Se la postazione di deposito NON è quella che sto considerando
													CONTINUE;														
												END_IF
											ELSE
												CONTINUE;
											END_IF
										END_FOR
									ELSE
										Debug_NessunaListaDaProcessare:=TRUE;
									END_IF
									
									(* Se nessuna Postazione Ha una lista in esecuzione Vado a cercare una postazione con lista da Eseguire *)
									(*IF PostazioneConListaInEsecuzione = 0 THEN
										IF WorkAreaProductionList^.Stato = LISTA_PROD_ASSENTE THEN	
											CONTINUE;								
										ELSIF WorkAreaProductionList^.Stato = LISTA_PROD_DA_ESEGUIRE OR WorkAreaProductionList^.Stato = LISTA_PROD_IN_ESECUZIONE THEN
											CASE WorkAreaProductionList^.PElement[WorkAreaState^[cwa].P].PElement.Typology OF
												LASTRA:
														WorkAreaManager^.State  := WAMANAGER_CICLO_LASTRA_WA_INIT;	(* Setto lo stato del WAMANAGER *)
														WADiDepositoFinale := cwa; //Memorizzo la Postazione FINALE di deposito
														RestoreCWA^ := TRUE;
														PreviousPWA^ := pwa;
														EXIT;
												FALDA:											
														WorkAreaManager^.State  := WAMANAGER_CICLO_FALDA_INIT;	(* Setto lo stato del WAMANAGER *)
														WADiDepositoFinale := cwa; //Memorizzo la Postazione FINALE di deposito
														RestoreCWA^ := TRUE;
														PreviousPWA^ := pwa;
														EXIT;
											END_CASE
										END_IF
									ELSE
										cwa := PostazioneConListaInEsecuzione;
										WADiDepositoFinale := cwa; //Memorizzo la Postazione FINALE di deposito
										IF WorkAreaState^[NumPostazioneDiPareggiatura].P > 1 THEN //Se ho la lastra depositata sulla tavola di pareggiatura, Riprendo dal Punto di pareggiatura
											IF PX_WorkArea[NumPostazioneDiPareggiatura] THEN //Se ho anche Presenza Fisica della lastra
												WorkAreaManager^.State  := WAMANAGER_CICLO_PAREGGIATURA_RUN;	(* Setto lo stato del WAMANAGER *)
												RIESEGUI_PAREGGIATURA := TRUE; //Forzo l'esecuzione della pareggiatura
											ELSE //Se non ho presenza Fisica della Lastra genero un errore
												Errore.Code := ErrWAM_FTC_OFF_PresenzaLastraPareggiatore; //Segnalo che la FTC non vede la presenza della lastra
											END_IF
										ELSE //Se non la lastra depositata sulla tavola di pareggiatura, Proseguo con la deposizione delle lastre sucessive
											CASE WorkAreaProductionList^.PElement[WorkAreaState^[cwa].P].PElement.Typology OF
												LASTRA:
														WorkAreaManager^.State  := WAMANAGER_CICLO_LASTRA_WA_INIT;	(* Setto lo stato del WAMANAGER *)
												FALDA:											
														WorkAreaManager^.State  := WAMANAGER_CICLO_FALDA_INIT;	(* Setto lo stato del WAMANAGER *)
											END_CASE
										END_IF
										RestoreCWA^ := TRUE;
										PreviousPWA^ := pwa;
										EXIT;
									END_IF*)								
							ELSE	
								;
							END_CASE
	{region "Ciclo falda"}
						WAMANAGER_CICLO_FALDA_INIT:	
							FALDA_INIT();						
															
						(*************************************************)
						(* Creo Missione FALDA *)	
						(*************************************************)
						WAMANAGER_CICLO_PRELIEVO_FALDA_RUN:	
							PREL_FALDA_RUN();

						WAMANAGER_CICLO_PRELIEVO_FALDA_END:
							PREL_FALDA_END();
							
							
						WAMANAGER_CICLO_DEPOSITO_FALDA_RUN:	
							DEP_FALDA_RUN();
							
						WAMANAGER_CICLO_DEPOSITO_FALDA_END:
							DEP_FALDA_END();
	{endregion}
	{region "Ciclo LASTRA DA PICK POINT"}														
						(*************************************************)
						(* Creo Missione LASTRA sul Punto di preievo *)	
						(*************************************************)
						WAMANAGER_CICLO_LASTRA_PP_INIT:
							LASTRA_PP_INIT();							
							
						WAMANAGER_CICLO_PRELIEVO_LASTRA_PP_RUN:
							PREL_LASTRA_PP_RUN();
							
						WAMANAGER_CICLO_PRELIEVO_LASTRA_PP_END:	
							PREL_LASTRA_PP_END();

						WAMANAGER_CICLO_DEPOSITO_LASTRA_PP_RUN:
							DEP_LASTRA_PP_RUN();
						
						WAMANAGER_CICLO_DEPOSITO_LASTRA_PP_END:
							DEP_LASTRA_PP_END();
	{endregion}	
	{region "Ciclo LASTRA DA WORKAREA"}
						(*************************************************)
						(* Creo Missione LASTRA Con Prelievo da WorkArea *)
						(*************************************************)
						WAMANAGER_CICLO_LASTRA_WA_INIT:
							LASTRA_WA_INIT();
							RestoreCWA^ := TRUE;
							PreviousPWA^ := pwa;
							EXIT;
							
						WAMANAGER_CICLO_PRELIEVO_LASTRA_WA_RUN:
							PREL_LASTRA_WA_RUN();
							RestoreCWA^ := TRUE;
							PreviousPWA^ := pwa;
							EXIT;
							
						WAMANAGER_CICLO_PRELIEVO_LASTRA_WA_END:
							PREL_LASTRA_WA_END();
							RestoreCWA^ := TRUE;
							PreviousPWA^ := pwa;
							EXIT;
							
						WAMANAGER_CICLO_DEPOSITO_LASTRA_SU_PAREGGIATORE_RUN:	
							DEP_PAREGGIATORE_RUN();			
												
						WAMANAGER_CICLO_DEPOSITO_LASTRA_SU_PAREGGIATORE_END:
							DEP_SU_PAREGGIATORE_END();
							
						WAMANAGER_CICLO_PAREGGIATURA_RUN:				
							CICLO_PAREGGIATURA_RUN();
	
						WAMANAGER_CICLO_PAREGGIATURA_END:
							CICLO_PAREGGIATURA_END();
							
						WAMANAGER_CICLO_PRELIEVO_LASTRA_DA_PAREGGIATORE_RUN:
							PREL_DA_PAREGGIATORE_RUN();
							
						WAMANAGER_CICLO_PRELIEVO_LASTRA_DA_PAREGGIATORE_END:
							PREL_DA_PAREGGIATORE_END();
				
						WAMANAGER_CICLO_DEPOSITO_LASTRA_WA_RUN:		
							DEP_LASTRA_WA_RUN();
							
						WAMANAGER_CICLO_DEPOSITO_LASTRA_WA_END:
							DEP_LASTRA_WA_END();
	{endregion}			

{endregion}		
					ELSE
						;
					END_CASE	//riferito al case WorkAreaManager^.State
				ELSE			// riferito all' IF prima del  case WorkAreaManager^.State
					RestoreCWA^ := TRUE;
					PreviousPWA^ := pwa;
					WorkAreaState^[cwa].State := WORKAREA_STATE_OCCUPIED_DISABLED;
					EXIT;
				END_IF			// riferito all' IF prima del case WorkAreaManager^.State	

(**********************************************************************************************************************************************************************************)
(**********************************************************************************************************************************************************************************)
			(* ******************************************************************************************************** *)
						(* GESTIONE (Nastratura) o (Veicolo per prelievo/deposito PALLET FINITI/CATASTE/FALDE) *)
			(* ******************************************************************************************************** *)
(**********************************************************************************************************************************************************************************)
(**********************************************************************************************************************************************************************************)
			(* Occupied + Worked *)
			WORKAREA_STATE_OCCUPIED_WORKED:
				IF WorkArea^[cwa].Enable = 1 THEN
					IF NOT WorkAreaState^[cwa].RefuseLGV THEN
						WorkAreaState^[cwa].State := WORKAREA_STATE_OCCUPIED_ENDED;
						(* Se NON BISOGNA eseguire la NASTRATURA *)		
						//IF Forming^[WorkAreaState^[cwa].F].Tape = 0 THEN
						//	WorkAreaState^[cwa].State := WORKAREA_STATE_OCCUPIED_ENDED;
						//(* Se BISOGNA eseguire la NASTRATURA *)	
						//ELSIF Forming^[WorkAreaState^[cwa].F].Tape = 1 THEN
						///	WorkAreaState^[cwa].State := WORKAREA_STATE_OCCUPIED_TAPING;
						//END_IF
					ELSIF WorkAreaState^[cwa].RefuseLGV AND WorkAreaState^[cwa].LGV_Req = 1 THEN
						WorkAreaState^[cwa].LGV_Req := NESSUNA_REQ_LGV;
						WorkAreaState^[cwa].LGV_GetIn_GetOut := NESSUNA_REQ_LGV;
					END_IF	
				ELSE
					WorkAreaState^[cwa].State := WORKAREA_STATE_OCCUPIED_WORKED_DISABLED;
				END_IF
	
			(* Occupied + Worked + Disabled *)
			WORKAREA_STATE_OCCUPIED_WORKED_DISABLED:
				WorkAreaState^[cwa].LGV_Req := NESSUNA_REQ_LGV;
				WorkAreaState^[cwa].LGV_GetIn_GetOut := NESSUNA_REQ_LGV;
				IF WorkArea^[cwa].Enable = 1 THEN
					WorkAreaState^[cwa].State := WORKAREA_STATE_OCCUPIED_WORKED;
				ELSE
					;
				END_IF
	
			(* Occupied + Taping *)
			WORKAREA_STATE_OCCUPIED_TAPING:
				WorkAreaState^[cwa].LGV_Req := NESSUNA_REQ_LGV;
				WorkAreaState^[cwa].LGV_GetIn_GetOut := NESSUNA_REQ_LGV;
				IF WorkArea^[cwa].Enable = 1 THEN
					IF WorkAreaState^[cwa].LGV_Req = 0 AND  WorkAreaState^[cwa].LGV_ReqAbort THEN
						WorkAreaState^[cwa].State := WORKAREA_STATE_OCCUPIED_WORKING;
						WorkAreaState^[cwa].LGV_ReqAbort := FALSE;
					ELSE
						//IF WorkArea^[cwa].Taped = 1 OR Forming^[WorkAreaState^[cwa].F].Tape = 0 THEN
						//	WorkAreaState^[cwa].State := WORKAREA_STATE_OCCUPIED_TAPED;
						//END_IF
					END_IF	
				ELSE
					WorkAreaState^[cwa].State := WORKAREA_STATE_OCCUPIED_TAPING_DISABLED;
				END_IF
	
			(* Occupied + Taping + Disabled *)
			WORKAREA_STATE_OCCUPIED_TAPING_DISABLED:
				IF WorkArea^[cwa].Enable = 1 THEN
					WorkAreaState^[cwa].State := WORKAREA_STATE_OCCUPIED_TAPING;
				ELSE
					;
				END_IF
	
			(* Occupied + Taped *)
			WORKAREA_STATE_OCCUPIED_TAPED:
				IF WorkArea^[cwa].Enable = 1 THEN
					WorkAreaState^[cwa].State := WORKAREA_STATE_OCCUPIED_ENDED;
				ELSE
					WorkAreaState^[cwa].State := WORKAREA_STATE_OCCUPIED_TAPED_DISABLED;
				END_IF
	
			(* Occupied + Taped + Disabled *)
			WORKAREA_STATE_OCCUPIED_TAPED_DISABLED:
				WorkAreaState^[cwa].LGV_Req := NESSUNA_REQ_LGV;
				WorkAreaState^[cwa].LGV_GetIn_GetOut := NESSUNA_REQ_LGV;
				IF WorkArea^[cwa].Enable = 1 THEN
					WorkAreaState^[cwa].State := WORKAREA_STATE_OCCUPIED_TAPED;
				ELSE
					;
				END_IF
	
			(* Occupied + Ended *)
			WORKAREA_STATE_OCCUPIED_ENDED:
				IF WorkArea^[cwa].Enable = 1 THEN
					IF WorkAreaState^[cwa].LGV_Req = NESSUNA_REQ_LGV AND  WorkAreaState^[cwa].LGV_ReqAbort THEN
						WorkAreaState^[cwa].State := WORKAREA_STATE_OCCUPIED_WORKING;
						WorkAreaState^[cwa].LGV_ReqAbort := FALSE;
					ELSIF WorkArea^[cwa].Typology = TYPOLOGY_PALLET	OR WorkArea^[cwa].Typology = TYPOLOGY_STACK AND NOT PX_WorkArea[cwa] THEN
						WorkAreaState^[cwa].State := WORKAREA_STATE_OCCUPIED_LGVREQ;
					END_IF	
				ELSE
					WorkAreaState^[cwa].State := WORKAREA_STATE_OCCUPIED_ENDED_DISABLED;
				END_IF
	
			(* Occupied + Ended + Disabled *)
			WORKAREA_STATE_OCCUPIED_ENDED_DISABLED:
				IF WorkArea^[cwa].Enable = 1 THEN
					WorkAreaState^[cwa].State := WORKAREA_STATE_OCCUPIED_ENDED;
				ELSE
					;
				END_IF
			(* Occupied + LgvReq *)
			WORKAREA_STATE_OCCUPIED_LGVREQ:
				IF WorkArea^[cwa].Enable = 1 THEN
					//IF Forming^[WorkAreaState^[cwa].F].Tape = 1 AND WorkArea^[cwa].Taped < 1 THEN
					//	WorkArea^[cwa].LGV_Req := NESSUNA_REQ_LGV;
					//	WorkArea^[cwa].LGV_GetIn_GetOut := NESSUNA_REQ_LGV;
					//	WorkArea^[cwa].LGV_ReqAbort := FALSE;
					//	WorkAreaState^[cwa].State := WORKAREA_STATE_OCCUPIED_WORKED;
					//	EXIT;
					//END_IF
					IF WorkAreaState^[cwa].LGV_ReqAbort AND WorkAreaState^[cwa].LGV_Req = NESSUNA_REQ_LGV THEN
						WorkAreaState^[cwa].LGV_Req 			:= NESSUNA_REQ_LGV;
						WorkAreaState^[cwa].LGV_GetIn_GetOut 	:= NESSUNA_REQ_LGV;
					ELSIF (NOT WorkAreaState^[cwa].LGV_ReqAbort AND WorkAreaState^[cwa].LGV_Req = NESSUNA_REQ_LGV) AND WorkArea^[cwa].Typology = TYPOLOGY_PALLET THEN//gestione postazione a terra
						//IF Forming^[WorkAreaState^[cwa].F].PackXP[WorkAreaState^[cwa].P].Grip = -1 OR
						//	Forming^[WorkAreaState^[cwa].F].PackXN[WorkAreaState^[cwa].P].Grip = -1 THEN
							(* Faccio la richiesta all'LGV di Tipo: PRELIEVO *)
						//	WorkArea^[cwa].LGV_Req := REQ_LGV;
						//	WorkArea^[cwa].LGV_GetIn_GetOut := REQ_PRELIEVO_LGV;  
						//ELSE
						//	WorkAreaState^[cwa].State := WORKAREA_STATE_OCCUPIED_WORKING;
						//	EXIT;
						//END_IF
						WorkAreaState^[cwa].LGV_Req 			:= NESSUNA_REQ_LGV;
						WorkAreaState^[cwa].LGV_GetIn_GetOut 	:= NESSUNA_REQ_LGV;  
					ELSIF (NOT WorkAreaState^[cwa].LGV_ReqAbort AND WorkAreaState^[cwa].LGV_Req = NESSUNA_REQ_LGV) AND WorkArea^[cwa].Typology = TYPOLOGY_BUNDLE THEN//gestione bundle
						WorkAreaState^[cwa].LGV_Req 			:= NESSUNA_REQ_LGV;
						WorkAreaState^[cwa].LGV_GetIn_GetOut 	:= NESSUNA_REQ_LGV;
						WorkAreaState^[cwa].State 				:= WORKAREA_STATE_FREE_WORKING;
					ELSE
						WorkAreaState^[cwa].LGV_Req := REQ_LGV;
						WorkAreaState^[cwa].LGV_GetIn_GetOut := REQ_PRELIEVO_LGV_PIENO;
					END_IF	
				ELSE
					WorkAreaState^[cwa].State := WORKAREA_STATE_OCCUPIED_LGVREQ_DISABLED;				
				END_IF
	
			(* Occupied + LgvReq + Disabled *)
			WORKAREA_STATE_OCCUPIED_LGVREQ_DISABLED:
				WorkAreaState^[cwa].LGV_Req := NESSUNA_REQ_LGV;
				WorkAreaState^[cwa].LGV_GetIn_GetOut := NESSUNA_REQ_LGV;
				IF WorkArea^[cwa].Enable = 1 THEN
					WorkAreaState^[cwa].State := WORKAREA_STATE_OCCUPIED_LGVREQ;
				ELSE
					;
				END_IF

			{Region "GESTIONE LGV non USATE"}	
			(* Occupied + LgvIn  - NOT USED !!!!!!!!!!!*)
			WORKAREA_STATE_OCCUPIED_LGVIN:
				IF WorkArea^[cwa].Enable = 1 THEN
					;
				ELSE
					;
				END_IF	
			(* Occupied + LgvIn + Disabled  - NOT USED !!!!!!!!!!!*)
			WORKAREA_STATE_OCCUPIED_LGVIN_DISABLED:
				IF WorkArea^[cwa].Enable = 1 THEN
					;
				ELSE
					;
				END_IF
			(* Occupied + LgvEnd  - NOT USED !!!!!!!!!!!*)
			WORKAREA_STATE_OCCUPIED_LGVEND:
				IF WorkArea^[cwa].Enable = 1 THEN
					;
				ELSE
					;
				END_IF
			(* Occupied + LgvIn + Disabled - NOT USED !!!!!!!!!!! *)
			WORKAREA_STATE_OCCUPIED_LGVEND_DISABLED:
				IF WorkArea^[cwa].Enable = 1 THEN
					;
				ELSE
					;
				END_IF
			{endregion}


			(* FREE + LgvReq *)
			WORKAREA_STATE_FREE_LGVREQ:
				IF WorkArea^[cwa].Enable = 1 THEN
					IF WorkAreaState^[cwa].LGV_ReqAbort AND WorkAreaState^[cwa].LGV_Req = NESSUNA_REQ_LGV THEN
						WorkAreaState^[cwa].LGV_Req := NESSUNA_REQ_LGV;
						WorkAreaState^[cwa].LGV_GetIn_GetOut := NESSUNA_REQ_LGV;
					ELSIF (NOT WorkAreaState^[cwa].LGV_ReqAbort AND WorkAreaState^[cwa].LGV_Req = NESSUNA_REQ_LGV) AND WorkArea^[cwa].Typology = TYPOLOGY_PALLET THEN
						WorkAreaState^[cwa].State := WORKAREA_STATE_OCCUPIED_WORKING;

					ELSE
						WorkAreaState^[cwa].LGV_Req 			:= REQ_LGV;
						WorkAreaState^[cwa].LGV_GetIn_GetOut 	:= REQ_DEPOSITO_LGV_VUOTO;
					END_IF	
				ELSE
					WorkAreaState^[cwa].State := WORKAREA_STATE_FREE_LGVREQ_DISABLED;				
				END_IF
	

			(* FREE + LgvReq + Disabled *)
			WORKAREA_STATE_FREE_LGVREQ_DISABLED:
				IF WorkArea^[cwa].Enable = 1 THEN
					WorkAreaState^[cwa].State := WORKAREA_STATE_FREE_LGVREQ;
				ELSE
					WorkAreaState^[cwa].LGV_Req 			:= NESSUNA_REQ_LGV;
					WorkAreaState^[cwa].LGV_GetIn_GetOut 	:= NESSUNA_REQ_LGV;
				END_IF

			(* Error *)
			WORKAREA_STATE_ERROR:
				;
	
		ELSE		//riferito al WorkAreaState^[cwa].State								
			(* Stato Errato. viene Forzato lo stato di errore. Non dovrebbe MAI accadere *)
			WorkAreaState^[cwa].State := WORKAREA_STATE_ERROR;
				
		END_CASE;  //riferito al WorkAreaState^[cwa].State
	
	END_FOR			// riferito a FOR pwa:=1 TO MAXAREA DO

END_IF 				// riferito a IF WaitPositionRequest > 0 AND

//TFPalletizerWorkAreaManagerTF := TRUE;

ACTION CICLO_PAREGGIATURA_END:
WorkAreaProductionList^[cwa].PElementList[ElList].Pareggiatura := PAREGGIATURA_ESEGUITA;
WorkAreaManager^.State := WAMANAGER_NOP;
RestoreCWA^ := TRUE;
PreviousPWA^ := pwa;
RETURN;//EXIT;

(* Mission^.PPlace	:= WADiDepositoFinale; (* valorizzo il punto di deposito *)
Mission^.PPick	:= INT_TO_UINT(NumPostazioneDiPareggiatura); (* valorizzo il punto di prelievo *)

NLastraDaPrelevare := WorkAreaState^[Mission^.PPick].P-1;
(* Il Valore di P indica il pacco da depositare, quindi se P-1 = TERMINATORE devo prelevare P-2 *)
IF Forming^[WorkAreaState^[Mission^.PPick].F].PElement[WorkAreaState^[Mission^.PPick].P].Typology = TERMINATORE THEN
	NLastraDaPrelevare := WorkAreaState^[Mission^.PPick].P-2;  							
END_IF

Mission^.TPick 	:= TPICK_LASTRA;	// Assegno il tipo di Prelievo
Mission^.XDim 	:= WorkAreaProductionList^[cwa].PElement[WorkAreaState^[cwa].P].PElement.XDim; 	// Assegno la dimensione X del pacco presente nel punto di prelievo designato
Mission^.YDim 	:= WorkAreaProductionList^[cwa].PElement[WorkAreaState^[cwa].P].PElement.YDim; 	// Assegno la dimensione Y del pacco presente nel punto di prelievo designato
Mission^.ZDim 	:= WorkAreaProductionList^[cwa].PElement[WorkAreaState^[cwa].P].PElement.ZDim; 	// Assegno la dimensione Z del pacco presente nel punto di prelievo designato



(* Assegnazione quote alla Missione *)
TFWAM_CreaMissione_PrelLastraDaWA(NPosInLavoro				:= Mission^.PPick, //Numero Postazione di depositio
									Angolo_Deposito 		:= Forming^[WorkAreaState^[Mission^.PPick].F].PElement[NLastraDaPrelevare].J, //Angolo di deposito dell'elemento
									PosizioneAttuale_X      := ModuleAX_X^.Ax^.Status.ActPosition, //Posizione attuale asse X
									TipologiaTraiettoria    := Forming^[WorkAreaState^[Mission^.PPick].F].PElement[NLastraDaPrelevare].Trajectory,
									
									Quota_PostX				:= WorkArea^[Mission^.PPick].X, //Quota X Postazione
									Quota_PostY				:= WorkArea^[Mission^.PPick].Y, //Quota Y Postazione
									Quota_PostZ				:= WorkArea^[Mission^.PPick].Z, //Quota Z Postazione
									Quota_PostJ				:= WorkArea^[Mission^.PPick].J, //Quota J Postazione
									
									Offset_Postazione_X 	:= WorkAreaOffset^[Mission^.PPick].X, //Offset X Postazione
									Offset_Postazione_Y 	:= WorkAreaOffset^[Mission^.PPick].Y, //Offset Y Postazione
									Offset_Postazione_Z 	:= WorkAreaOffset^[Mission^.PPick].Z, //Offset Z Postazione
									Offset_Postazione_J 	:= WorkAreaOffset^[Mission^.PPick].J, //Offset J Postazione
									
									Pallet_DimX				:= Forming^[WorkAreaState^[Mission^.PPick].F].Pallet.XDim, //Dimensione X Pallet
									Pallet_DimY				:= Forming^[WorkAreaState^[Mission^.PPick].F].Pallet.YDim, //Dimensione Y Pallet
									Pallet_DimZ				:= Forming^[WorkAreaState^[Mission^.PPick].F].Pallet.ZDim, //Dimensione Z Pallet
									
									Offset_Pallet_X_0		:= Forming^[WorkAreaState^[Mission^.PPick].F].Pallet.OFSDE_X0, //Offset X Pallet o Casse
									Offset_Pallet_Y_0		:= Forming^[WorkAreaState^[Mission^.PPick].F].Pallet.OFSDE_Y0, //Offset Y Pallet o Casse 
									Offset_Pallet_Z_0		:= Forming^[WorkAreaState^[Mission^.PPick].F].Pallet.OFSDE_Z0, //Offset Z Pallet o Casse + è grande + il deposito si distanzia dal supporto
									Offset_Pallet_J_0		:= Forming^[WorkAreaState^[Mission^.PPick].F].Pallet.OFSDE_J0, //Offset J Pallet o Casse + è grande + la lastra sarà inclinata verso l'angolo crescente
									
									Offset_Pallet_X_90		:= Forming^[WorkAreaState^[Mission^.PPick].F].Pallet.OFSDE_X90, //Offset X Pallet lato 0-90 
									Offset_Pallet_Y_90		:= Forming^[WorkAreaState^[Mission^.PPick].F].Pallet.OFSDE_Y90, //Offset Y Pallet lato 0-90 + è grande + il deposito si distanzia dal supporto
									Offset_Pallet_Z_90		:= Forming^[WorkAreaState^[Mission^.PPick].F].Pallet.OFSDE_Z90, //Offset Z Pallet lato 0-90 + è grande + il deposito si distanzia dal supporto
									Offset_Pallet_J_90		:= Forming^[WorkAreaState^[Mission^.PPick].F].Pallet.OFSDE_J90, //Offset J Pallet lato 0-90 + è grande + la lastra sarà inclinata in fase di deposito
									
									Offset_Pallet_X_180		:= Forming^[WorkAreaState^[Mission^.PPick].F].Pallet.OFSDE_X180, //Offset X Pallet lato 90-180
									Offset_Pallet_Y_180		:= Forming^[WorkAreaState^[Mission^.PPick].F].Pallet.OFSDE_Y180, //Offset Y Pallet lato 90-180 + è grande + il deposito si distanzia dal supporto
									Offset_Pallet_Z_180		:= Forming^[WorkAreaState^[Mission^.PPick].F].Pallet.OFSDE_Z180, //Offset Z Pallet lato 90-180 + è grande + il deposito si distanzia dal supporto
									Offset_Pallet_J_180		:= Forming^[WorkAreaState^[Mission^.PPick].F].Pallet.OFSDE_J180, //Offset J Pallet lato 90-180 + è grande + la lastra sarà inclinata in fase di deposito
									
									Quota_FormaturaX 		:= Forming^[WorkAreaState^[Mission^.PPick].F].PElement[NLastraDaPrelevare].X, //Quota Deposito X da Formatura
									Quota_FormaturaY 		:= Forming^[WorkAreaState^[Mission^.PPick].F].PElement[NLastraDaPrelevare].Y, //Quota Deposito Y da Formatura
									Quota_FormaturaZ 		:= Forming^[WorkAreaState^[Mission^.PPick].F].PElement[NLastraDaPrelevare].Z, //Quota Deposito Z da Formatura
									Quota_FormaturaJ 		:= Forming^[WorkAreaState^[Mission^.PPick].F].PElement[NLastraDaPrelevare].J, //Quota Deposito Z da Formatura
									
									Distanza_ApproccioFormaturaX 		:= Forming^[WorkAreaState^[Mission^.PPick].F].PElement[NLastraDaPrelevare].AX, //Quota Deposito X da Formatura
									Distanza_ApproccioFormaturaY 		:= Forming^[WorkAreaState^[Mission^.PPick].F].PElement[NLastraDaPrelevare].AY, //Quota Deposito Y da Formatura
									Distanza_ApproccioFormaturaZ 		:= Forming^[WorkAreaState^[Mission^.PPick].F].PElement[NLastraDaPrelevare].AZ, //Quota Deposito Z da Formatura
									Distanza_ApproccioFormaturaJ 		:= Forming^[WorkAreaState^[Mission^.PPick].F].PElement[NLastraDaPrelevare].AJ, //Quota Deposito Z da Formatura
									
									Quota_DestX 			=> Mission^.XPick, //Quota DESTINAZIONE X
									Quota_DestY 			=> Mission^.YPick, //Quota DESTINAZIONE Y
									Quota_DestZ 			=> Mission^.ZPick, //Quota DESTINAZIONE Z
									Quota_DestJ 			=> Mission^.JPick, //Quota DESTINAZIONE J	
									
									Quota_ApproccioDestX 	=> Mission^.XPickApproach, //Quota APPROCCIO di DESTINAZIONE X
									Quota_ApproccioDestY 	=> Mission^.YPickApproach, //Quota APPROCCIO di DESTINAZIONE Y
									Quota_ApproccioDestZ 	=> Mission^.ZPickApproach, //Quota APPROCCIO di DESTINAZIONE Z
									Quota_ApproccioDestJ 	=> Mission^.JPickApproach);//Quota APPROCCIO di DESTINAZIONE J	

IF TFWAM_CreaMissione_PrelLastraDaWA.Errore.Code > 0 THEN
		Errore.Code := TFWAM_CreaMissione_PrelLastraDaWA.Errore;
		WorkAreaManager^.State 	:= WAMANAGER_NOP;	// setto lo stato del WAMANAGER
		EXIT;
END_IF
	
(* Valorizzazione quote di deposito Ciclo Lastra *)
TFWAM_CreaMissione_DepLastraDaWA(NPosInLavoro			:= Mission^.PPlace, //Numero Postazione di depositio
									Angolo_Deposito 		:= Forming^[WorkAreaState^[Mission^.PPlace].F].PElement[WorkAreaState^[Mission^.PPlace].P].J, //Angolo di deposito dell'elemento
									PosizioneAttuale_X      := ModuleAX_X^.Ax^.Status.ActPosition, //Posizione attuale asse X
									TipologiaTraiettoria    := Forming^[WorkAreaState^[cwa].F].PElement[WorkAreaState^[cwa].P].Trajectory,
										
									Quota_PostX				:= WorkArea^[Mission^.PPlace].X, //Quota X Postazione
									Quota_PostY				:= WorkArea^[Mission^.PPlace].Y, //Quota Y Postazione
									Quota_PostZ				:= WorkArea^[Mission^.PPlace].Z, //Quota Z Postazione
									Quota_PostJ				:= WorkArea^[Mission^.PPlace].J, //Quota J Postazione
									
									Offset_Postazione_X 	:= WorkAreaOffset^[Mission^.PPlace].X, //Offset X Postazione
									Offset_Postazione_Y 	:= WorkAreaOffset^[Mission^.PPlace].Y, //Offset Y Postazione
									Offset_Postazione_Z 	:= WorkAreaOffset^[Mission^.PPlace].Z, //Offset Z Postazione
									Offset_Postazione_J 	:= WorkAreaOffset^[Mission^.PPlace].J, //Offset J Postazione
									
									Pallet_DimX				:= Forming^[WorkAreaState^[Mission^.PPlace].F].Pallet.XDim, //Dimensione X Pallet
									Pallet_DimY				:= Forming^[WorkAreaState^[Mission^.PPlace].F].Pallet.YDim, //Dimensione Y Pallet
									Pallet_DimZ				:= Forming^[WorkAreaState^[Mission^.PPlace].F].Pallet.ZDim, //Dimensione Z Pallet
									
									Offset_Pallet_X_0		:= Forming^[WorkAreaState^[Mission^.PPlace].F].Pallet.OFSDE_X0, //Offset X Pallet o Casse
									Offset_Pallet_Y_0		:= Forming^[WorkAreaState^[Mission^.PPlace].F].Pallet.OFSDE_Y0, //Offset Y Pallet o Casse 
									Offset_Pallet_Z_0		:= Forming^[WorkAreaState^[Mission^.PPlace].F].Pallet.OFSDE_Z0, //Offset Z Pallet o Casse + è grande + il deposito si distanzia dal supporto
									Offset_Pallet_J_0		:= Forming^[WorkAreaState^[Mission^.PPlace].F].Pallet.OFSDE_J0, //Offset J Pallet o Casse + è grande + la lastra sarà inclinata verso l'angolo crescente
									
									Offset_Pallet_X_90		:= Forming^[WorkAreaState^[Mission^.PPlace].F].Pallet.OFSDE_X90, //Offset X Pallet lato 0-90 
									Offset_Pallet_Y_90		:= Forming^[WorkAreaState^[Mission^.PPlace].F].Pallet.OFSDE_Y90, //Offset Y Pallet lato 0-90 + è grande + il deposito si distanzia dal supporto
									Offset_Pallet_Z_90		:= Forming^[WorkAreaState^[Mission^.PPlace].F].Pallet.OFSDE_Z90, //Offset Z Pallet lato 0-90 + è grande + il deposito si distanzia dal supporto
									Offset_Pallet_J_90		:= Forming^[WorkAreaState^[Mission^.PPlace].F].Pallet.OFSDE_J90, //Offset J Pallet lato 0-90 + è grande + la lastra sarà inclinata in fase di deposito
									
									Offset_Pallet_X_180		:= Forming^[WorkAreaState^[Mission^.PPlace].F].Pallet.OFSDE_X180, //Offset X Pallet lato 90-180
									Offset_Pallet_Y_180		:= Forming^[WorkAreaState^[Mission^.PPlace].F].Pallet.OFSDE_Y180, //Offset Y Pallet lato 90-180 + è grande + il deposito si distanzia dal supporto
									Offset_Pallet_Z_180		:= Forming^[WorkAreaState^[Mission^.PPlace].F].Pallet.OFSDE_Z180, //Offset Z Pallet lato 90-180 + è grande + il deposito si distanzia dal supporto
									Offset_Pallet_J_180		:= Forming^[WorkAreaState^[Mission^.PPlace].F].Pallet.OFSDE_J180, //Offset J Pallet lato 90-180 + è grande + la lastra sarà inclinata in fase di deposito
									
									Quota_FormaturaX 		:= Forming^[WorkAreaState^[Mission^.PPlace].F].PElement[WorkAreaState^[Mission^.PPlace].P].X, //Quota Deposito X da Formatura
									Quota_FormaturaY 		:= Forming^[WorkAreaState^[Mission^.PPlace].F].PElement[WorkAreaState^[Mission^.PPlace].P].Y, //Quota Deposito Y da Formatura
									Quota_FormaturaZ 		:= Forming^[WorkAreaState^[Mission^.PPlace].F].PElement[WorkAreaState^[Mission^.PPlace].P].Z, //Quota Deposito Z da Formatura
									Quota_FormaturaJ 		:= Forming^[WorkAreaState^[Mission^.PPlace].F].PElement[WorkAreaState^[Mission^.PPlace].P].J, //Quota Deposito Z da Formatura
									
									Distanza_ApproccioFormaturaX 		:= Forming^[WorkAreaState^[Mission^.PPlace].F].PElement[WorkAreaState^[Mission^.PPlace].P].AX, //Quota Deposito X da Formatura
									Distanza_ApproccioFormaturaY 		:= Forming^[WorkAreaState^[Mission^.PPlace].F].PElement[WorkAreaState^[Mission^.PPlace].P].AY, //Quota Deposito Y da Formatura
									Distanza_ApproccioFormaturaZ 		:= Forming^[WorkAreaState^[Mission^.PPlace].F].PElement[WorkAreaState^[Mission^.PPlace].P].AZ, //Quota Deposito Z da Formatura
									Distanza_ApproccioFormaturaJ 		:= Forming^[WorkAreaState^[Mission^.PPlace].F].PElement[WorkAreaState^[Mission^.PPlace].P].AJ, //Quota Deposito Z da Formatura
									
									Quota_DestX 			=> Mission^.XPlace, //Quota DESTINAZIONE X
									Quota_DestY 			=> Mission^.YPlace, //Quota DESTINAZIONE Y
									Quota_DestZ 			=> Mission^.ZPlace, //Quota DESTINAZIONE Z
									Quota_DestJ 			=> Mission^.JPlace, //Quota DESTINAZIONE J	
									
									Quota_ApproccioDestX 	=> Mission^.XPlaceApproach, //Quota APPROCCIO di DESTINAZIONE X
									Quota_ApproccioDestY 	=> Mission^.YPlaceApproach, //Quota APPROCCIO di DESTINAZIONE Y
									Quota_ApproccioDestZ 	=> Mission^.ZPlaceApproach, //Quota APPROCCIO di DESTINAZIONE Z
									Quota_ApproccioDestJ 	=> Mission^.JPlaceApproach);//Quota APPROCCIO di DESTINAZIONE J	

IF TFWAM_CreaMissione_PrelLastraDaWA.Errore.Code > 0 THEN
		Errore.Code := TFWAM_CreaMissione_PrelLastraDaWA.Errore;
		EXIT;
ELSE
	WorkAreaManager^.State 	:= WAMANAGER_CICLO_PRELIEVO_LASTRA_DA_PAREGGIATORE_RUN;	// setto lo stato del WAMANAGER
	RestoreCWA^ := TRUE;
	PreviousPWA^ := pwa;
	EXIT;
END_IF*)
END_ACTION

ACTION CICLO_PAREGGIATURA_RUN:
IF Mission^.State = MISSION_STATE_PAREGGIATURA_RUN THEN
	;
ELSIF Mission^.State = MISSION_STATE_PAREGGIATURA_END OR WorkAreaProductionList^[cwa].PElementList[ElList].Pareggiatura = PAREGGIATURA_DA_ESEGUIRE THEN
	;
ELSIF Mission^.State = MISSION_STATE_ERROR THEN
	;
END_IF
END_ACTION

ACTION DEP_FALDA_END:
(* Aggiorno la struttura lastre della postazione *)
WorkAreaState^[Mission^.PPlace].Slab[WorkAreaState^[Mission^.PPlace].P]  := Mission^.Slab;
(* Incremento WorkArea^[cwa].P (P=P+1) *)
WorkAreaState^[Mission^.PPlace].P := WorkAreaState^[Mission^.PPlace].P + 1;
WorkAreaProductionList^[Mission^.PPlace].PElementList[ElList].Stato := ELEMENTO_ELABORATO; //Dichiaro che l'elemnto della lista è stato elaborato
WorkAreaManager^.State := WAMANAGER_NOP;
RestoreCWA^ := TRUE;
PreviousPWA^ := pwa;
RETURN;//EXIT;
END_ACTION

ACTION DEP_FALDA_RUN:
IF Mission^.State = MISSION_STATE_DEPOSITO_FALDA_RUN THEN
	;
ELSIF Mission^.State = MISSION_STATE_DEPOSITO_FALDA_END THEN
	WorkAreaManager^.State 	:= WAMANAGER_CICLO_DEPOSITO_FALDA_END;	// setto lo stato del WAMANAGER
	RETURN;//EXIT;
ELSIF Mission^.State = MISSION_STATE_ERROR THEN
	;
END_IF
END_ACTION

ACTION DEP_LASTRA_PP_END:
(* Se era settata la velocità lenta di deposito pacco, questa viene resettata *)
IF WorkAreaState^[Mission^.PPlace].Slow = 1 THEN
	WorkAreaState^[Mission^.PPlace].Slow := 0;
	DepositoPaccoInLenta := FALSE;
END_IF
(* Aggiorno la struttura lastre della postazione *)
WorkAreaState^[Mission^.PPlace].Slab[WorkAreaState^[Mission^.PPlace].P]  := Mission^.Slab;
(* Incremento WorkArea^[cwa].P (P=P+1) *)
WorkAreaState^[Mission^.PPlace].P := WorkAreaState^[Mission^.PPlace].P + 1;

//IF HMI_AbilitaDepositoPaccoOrrizzontaleConTasteggio THEN
	(* Imposto lo stato dell' apprendimento *)
	CASE LatoDeposito OF			
		(*0:
			IF WorkAreaState^[Mission^.PPlace].Apprendimento.Y.Lato0.Stato <> APPRENDIMENTO_ESEGUITO THEN
				WorkAreaState^[Mission^.PPlace].Apprendimento.Y.Lato0.Stato := APPRENDIMENTO_ESEGUITO;
				WorkAreaState^[Mission^.PPlace].Apprendimento.Y.Lato0.QuotaRilevata := ModuleAX_Y^.QuotaAsseLetturaTasteggio;
			ELSE
				WorkAreaState^[Mission^.PPlace].Apprendimento.Y.Lato0.QuotaRilevata := ModuleAX_Y^.QuotaAsseLetturaTasteggio;
			END_IF*)
		90:
			IF WorkAreaState^[Mission^.PPlace].Apprendimento.Z.Lato90.Stato <> APPRENDIMENTO_ESEGUITO THEN
				WorkAreaState^[Mission^.PPlace].Apprendimento.Z.Lato90.Stato 				:= APPRENDIMENTO_ESEGUITO;
				WorkAreaState^[Mission^.PPlace].Apprendimento.Z.Lato90.QuotaRilevata 		:= ModuleAX_Z^.QuotaAsseLetturaTasteggio;
				WorkAreaState^[Mission^.PPlace].Supporto.HMAX 	:=  MAX(WorkAreaState^[Mission^.PPlace].Supporto.HMAX,ModuleAX_Z^.QuotaAsseLetturaTasteggio);
				WorkAreaState^[Mission^.PPlace].H 				:=  ModuleAX_Z^.QuotaAsseLetturaTasteggio;
				WorkAreaState^[Mission^.PPlace].HPL 			:=  ModuleAX_Z^.QuotaAsseLetturaTasteggio;	 

			ELSE
				WorkAreaState^[Mission^.PPlace].Apprendimento.Z.Lato90.Stato 				:= 	APPRENDIMENTO_ESEGUITO;
				WorkAreaState^[Mission^.PPlace].Apprendimento.Z.Lato90.QuotaRilevata 		:=  ModuleAX_Z^.QuotaAsseLetturaTasteggio;
				WorkAreaState^[Mission^.PPlace].Supporto.HMAX 	:=  MAX(WorkAreaState^[Mission^.PPlace].Supporto.HMAX,ModuleAX_Z^.QuotaAsseLetturaTasteggio);
				WorkAreaState^[Mission^.PPlace].H 				:=  ModuleAX_Z^.QuotaAsseLetturaTasteggio;
				WorkAreaState^[Mission^.PPlace].HPL 			:=  ModuleAX_Z^.QuotaAsseLetturaTasteggio;	 

			END_IF
		(*180:
			IF WorkAreaState^[Mission^.PPlace].Apprendimento.Y.Lato180.Stato <> APPRENDIMENTO_ESEGUITO THEN
				WorkAreaState^[Mission^.PPlace].Apprendimento.Y.Lato180.Stato := APPRENDIMENTO_ESEGUITO;
				WorkAreaState^[Mission^.PPlace].Apprendimento.Y.Lato180.QuotaRilevata := ModuleAX_Y^.QuotaAsseLetturaTasteggio;
			ELSE
				WorkAreaState^[Mission^.PPlace].Apprendimento.Y.Lato180.QuotaRilevata := ModuleAX_Y^.QuotaAsseLetturaTasteggio;
			END_IF*)
	END_CASE
//END_IF
(* Controllo se la Pallettizzazione è TERMINATA *)
IF Forming^[WorkAreaState^[Mission^.PPlace].F].PElement[WorkAreaState^[Mission^.PPlace].P].Typology = TERMINATORE THEN
	WorkAreaManager^.State 	:= WAMANAGER_NOP;	// setto lo stato del WAMANAGER
	RestoreCWA^ := TRUE;
	PreviousPWA^ := Mission^.PPlace;
	RETURN;//EXIT;
ELSE
	WorkAreaManager^.State 	:= WAMANAGER_NOP;	// setto lo stato del WAMANAGER
	RestoreCWA^ := TRUE;
	PreviousPWA^ := Mission^.PPlace;
	RETURN;//EXIT;
END_IF
END_ACTION

ACTION DEP_LASTRA_PP_RUN:

IF Mission^.State = MISSION_STATE_DEPOSITO_LASTRA_PP_RUN THEN
	;
ELSIF Mission^.State = MISSION_STATE_DEPOSITO_LASTRA_PP_END THEN
	WorkAreaManager^.State 	:= WAMANAGER_CICLO_DEPOSITO_LASTRA_PP_END;
ELSIF Mission^.State = MISSION_STATE_ERROR THEN
	;
END_IF
END_ACTION

ACTION DEP_LASTRA_WA_END:

(* Se era settata la velocità lenta di deposito pacco, questa viene resettata *)
IF WorkAreaState^[Mission^.PPlace].Slow = 1 THEN
	WorkAreaState^[Mission^.PPlace].Slow := 0;
	DepositoPaccoInLenta := FALSE;
END_IF

(* Controllo se la Pallettizzazione è TERMINATA *)
IF Forming^[WorkAreaState^[Mission^.PPlace].F].PElement[WorkAreaState^[Mission^.PPlace].P].Typology = TERMINATORE THEN
	WorkAreaManager^.State 	:= WAMANAGER_NOP;	// setto lo stato del WAMANAGER
	WorkAreaProductionList^[Mission^.PPlace].PElementList[ElList].Stato := ELEMENTO_ELABORATO; //Dichiaro che l'elemento della lista è stato elaborato
ELSE
	WorkAreaManager^.State 	:= WAMANAGER_NOP;	// setto lo stato del WAMANAGER
	WorkAreaProductionList^[Mission^.PPlace].PElementList[ElList].Stato := ELEMENTO_ELABORATO; //Dichiaro che l'elemento della lista è stato elaborato
END_IF

(* Aggiorno la struttura lastre della postazione *)
WorkAreaState^[Mission^.PPlace].Slab[WorkAreaState^[Mission^.PPlace].P] := Mission^.Slab;
(* Incremento WorkArea^[cwa].P (P=P+1) *)
WorkAreaState^[Mission^.PPlace].P := WorkAreaState^[Mission^.PPlace].P + 1;

IF WorkAreaState^[Mission^.PPlace].Supporto.Tipologia = CAVALLETTO THEN 
		IF PosicionJDestino = 0 THEN 
			WorkAreaState^[Mission^.PPlace].P_Cava.HMI_NumeroPezziPresentiPostazione_A_Cavaleto := WorkAreaState^[Mission^.PPlace].P_Cava.HMI_NumeroPezziPresentiPostazione_A_Cavaleto +1 ;
		ELSIF PosicionJDestino = 180 THEN 	
			WorkAreaState^[Mission^.PPlace].P_Cava.HMI_NumeroPezziPresentiPostazione_B_Cavaleto := WorkAreaState^[Mission^.PPlace].P_Cava.HMI_NumeroPezziPresentiPostazione_B_Cavaleto +1 ;
		END_IF
END_IF
(* Imposto lo stato dell' apprendimento *)
CASE LatoDeposito OF			
	(*0:
		IF WorkAreaState^[Mission^.PPlace].Apprendimento.Y.Lato0.Stato <> APPRENDIMENTO_ESEGUITO THEN
			WorkAreaState^[Mission^.PPlace].Apprendimento.Y.Lato0.Stato := APPRENDIMENTO_ESEGUITO;
			WorkAreaState^[Mission^.PPlace].Apprendimento.Y.Lato0.QuotaRilevata := ModuleAX_Y^.QuotaAsseLetturaTasteggio;
		ELSE
			WorkAreaState^[Mission^.PPlace].Apprendimento.Y.Lato0.QuotaRilevata := ModuleAX_Y^.QuotaAsseLetturaTasteggio;
		END_IF*)
	90:
		IF WorkAreaState^[Mission^.PPlace].Apprendimento.Z.Lato90.Stato <> APPRENDIMENTO_ESEGUITO THEN
			WorkAreaState^[Mission^.PPlace].Apprendimento.Z.Lato90.Stato 				:= APPRENDIMENTO_ESEGUITO;
			WorkAreaState^[Mission^.PPlace].Apprendimento.Z.Lato90.QuotaRilevata 		:= ModuleAX_Z^.QuotaAsseLetturaTasteggio;
			WorkAreaState^[Mission^.PPlace].Supporto.HMAX 	:=  MAX(WorkAreaState^[Mission^.PPlace].Supporto.HMAX,ModuleAX_Z^.QuotaAsseLetturaTasteggio);
			WorkAreaState^[Mission^.PPlace].H 				:=  ModuleAX_Z^.QuotaAsseLetturaTasteggio;
			WorkAreaState^[Mission^.PPlace].HPL 			:=  ModuleAX_Z^.QuotaAsseLetturaTasteggio;	 

		ELSE
			WorkAreaState^[Mission^.PPlace].Apprendimento.Z.Lato90.Stato 				:= 	APPRENDIMENTO_ESEGUITO;
			WorkAreaState^[Mission^.PPlace].Apprendimento.Z.Lato90.QuotaRilevata 		:=  ModuleAX_Z^.QuotaAsseLetturaTasteggio;
			WorkAreaState^[Mission^.PPlace].Supporto.HMAX 	:=  MAX(WorkAreaState^[Mission^.PPlace].Supporto.HMAX,ModuleAX_Z^.QuotaAsseLetturaTasteggio);
			WorkAreaState^[Mission^.PPlace].H 				:=  ModuleAX_Z^.QuotaAsseLetturaTasteggio;
			WorkAreaState^[Mission^.PPlace].HPL 			:=  ModuleAX_Z^.QuotaAsseLetturaTasteggio;	 

		END_IF
	(*180:
		IF WorkAreaState^[Mission^.PPlace].Apprendimento.Y.Lato180.Stato <> APPRENDIMENTO_ESEGUITO THEN
			WorkAreaState^[Mission^.PPlace].Apprendimento.Y.Lato180.Stato := APPRENDIMENTO_ESEGUITO;
			WorkAreaState^[Mission^.PPlace].Apprendimento.Y.Lato180.QuotaRilevata := ModuleAX_Y^.QuotaAsseLetturaTasteggio;
		ELSE
			WorkAreaState^[Mission^.PPlace].Apprendimento.Y.Lato180.QuotaRilevata := ModuleAX_Y^.QuotaAsseLetturaTasteggio;
		END_IF*)
END_CASE


//RestoreCWA^ := TRUE;
//PreviousPWA^ := pwa;
WorkAreaManager^.State 	:= WAMANAGER_NOP;	// setto lo stato del WAMANAGER
END_ACTION

ACTION DEP_LASTRA_WA_RUN:
		
IF Mission^.State = MISSION_STATE_DEPOSITO_LASTRA_WA_RUN THEN
	WorkAreaManager^.State 	:= WAMANAGER_CICLO_DEPOSITO_LASTRA_WA_RUN;
ELSIF Mission^.State = MISSION_STATE_DEPOSITO_LASTRA_WA_END THEN
	WorkAreaManager^.State 	:= WAMANAGER_CICLO_DEPOSITO_LASTRA_WA_END;
ELSIF Mission^.State = MISSION_STATE_ERROR THEN
	;
END_IF
END_ACTION

ACTION DEP_PAREGGIATORE_RUN:
IF Mission^.State = MISSION_STATE_DEPOSITO_LASTRA_SU_PAREGGIATORE_RUN THEN
	;
ELSIF Mission^.State = MISSION_STATE_DEPOSITO_LASTRA_SU_PAREGGIATORE_END THEN
	WorkAreaManager^.State 	:= WAMANAGER_CICLO_DEPOSITO_LASTRA_SU_PAREGGIATORE_END;
ELSIF Mission^.State = MISSION_STATE_ERROR THEN
	;
END_IF
END_ACTION

ACTION DEP_SU_PAREGGIATORE_END:
(* Se era settata la velocità lenta di deposito pacco, questa viene resettata *)
IF WorkAreaState^[Mission^.PPlace].Slow = 1 THEN
	WorkAreaState^[Mission^.PPlace].Slow := 0;
	DepositoPaccoInLenta := FALSE;
END_IF
(* Aggiorno la struttura lastre della postazione *)
WorkAreaState^[Mission^.PPlace].Slab[WorkAreaState^[Mission^.PPlace].P]  := Mission^.Slab;
(* Incremento WorkArea^[cwa].P (P=P+1) *)
WorkAreaState^[Mission^.PPlace].P := WorkAreaState^[Mission^.PPlace].P + 1;

WorkAreaManager^.State 	:= WAMANAGER_CICLO_PAREGGIATURA_RUN;	// setto lo stato del WAMANAGER
RestoreCWA^ := TRUE;
PreviousPWA^ := pwa;
RETURN;//EXIT;
END_ACTION

ACTION DEP_SU_PAREGGIATORE_RUN:

END_ACTION

ACTION FALDA_INIT:
(* Nel caso si esca esca dal ciclo continuo a valutare la postazione in esame *)
RestoreCWA^ := TRUE;
PreviousPWA^ := pwa;
		
(* Creo Missione Falda *)
Mission^.PPick			:= ppick; 				(* valorizzo il punto di prelievo = workarea dove ho valutato la presenza delle falde *)
Mission^.PPlace			:= cwa;					(* valorizzo il punto di deposito = workarea dove ho valutato di depositare la falda *)						
IF TIPO_MAGAZZINO_FALDE = MAGAZZINO_FALDE_IN_PP THEN 		(* Se il magazzino delle falde è PickPoint *)
	IF WorkPickPoint^[Mission^.PPick].Tipologia = MAGAZZINO_FALDE THEN
		
		CASE WorkPickPointState^[Mission^.PPick].Element.TypologyCode OF //Layer^[WorkPickPointStoreState^[Mission^.PPick].Code].Tipologia OF
			FALDA_CARTONE :
				Mission^.TPick 		:= TPICK_LAY_VENTOSE;			(* valorizzo la tipologia di prelievo = tipo prelievo falda *)
			FALDA_POLISTIROLO :
				IF Forming^[WorkAreaState^[Mission^.PPlace].F].AuxAttr.1 = 1 THEN
					Mission^.TPick	:= TPICK_LAY_ARPIONI;			(* valorizzo la tipologia di prelievo = tipo prelievo falda *)
				ELSE
					Mission^.TPick	:= TPICK_LAY_VENTOSE;			(* valorizzo la tipologia di prelievo = tipo prelievo falda *)
				END_IF
		ELSE
			Mission^.TPick 	:= TPICK_NOT_DEFINED;					(* valorizzo la tipologia di prelievo = tipo prelievo falda	*)
			Errore.Code 	:= ErrWAM_TipologiaFaldaNONRiconosciuta;(* E' stata impostata una tipologia di falda non prevista per l'impianto *)
			RETURN;//EXIT;
		END_CASE
	ELSE
		Errore.Code := ErrWAM_PickPoint_NoMagazzinoFalde;(*Errore, Il Pick Point, non è di tipo Magazzino Falde *)
		RETURN;//EXIT;
	END_IF
	Mission^.XPick			:= WorkPickPoint^[Mission^.PPick].X + (Layer^[WorkPickPointState^[WorkPickPoint^[Mission^.PPick].ID].Code].XDim/2); (* valorizzo la quota X di prelievo *)
	Mission^.YPick			:= WorkPickPoint^[Mission^.PPick].Y + (Layer^[WorkPickPointState^[WorkPickPoint^[Mission^.PPick].ID].Code].YDim/2); (* valorizzo la quota Y di prelievo *)
	Mission^.ZPick			:= WorkPickPoint^[Mission^.PPick].Z; (* in questo modo LA LENTA va sempre fino a zero...mi fermo al raggiungimento dell'intervento dei tastatori *)
	Mission^.JPick			:= WorkPickPoint^[Mission^.PPick].J;
ELSIF TIPO_MAGAZZINO_FALDE = MAGAZZINO_FALDE_IN_WA THEN 	(* Se il magazzino delle falde è una WorkArea *)
	(*IF WorkArea^[Mission^.PPick].Typology = TYPOLOGY_LAYER THEN
		CASE WorkAreaState^[Mission^.PPick].Typology_Description OF
			FALDA_CARTONE :
				Mission^.TPick 			:= TPICK_LAY_VENTOSE;			(* valorizzo la tipologia di prelievo = tipo prelievo falda *)
			FALDA_POLISTIROLO :
				IF Forming^[WorkAreaState^[Mission^.PPlace].F].AuxAttr.1 = 1 THEN
					Mission^.TPick 		:= TPICK_LAY_ARPIONI;		(* valorizzo la tipologia di prelievo = tipo prelievo falda *)
				ELSE
					Mission^.TPick 		:= TPICK_LAY_VENTOSE;		(* valorizzo la tipologia di prelievo = tipo prelievo falda *)
				END_IF
		ELSE
			Mission^.TPick 				:= TPICK_NOT_DEFINED;			(* valorizzo la tipologia di prelievo = tipo prelievo falda	*)
			Errore.Code := ErrWAM_TipologiaFaldaNONRiconosciuta; 	(* E' stata impostata una tipologia di falda non prevista per l'impianto *)
			EXIT;
		END_CASE
	ELSE
		Errore.Code := ErrWAM_WorkArea_NoMagazzinoFalde; (* Errore, la WorkArea non è di tipo Magazzino Falde *)
		EXIT;
	END_IF*)
	
	IF Forming^[WorkAreaState^[Mission^.PPlace].F].AuxAttr.1 = 1 THEN
		Mission^.TPick 		:= TPICK_LAY_ARPIONI;		(* valorizzo la tipologia di prelievo = tipo prelievo falda *)
	ELSE
		Mission^.TPick 		:= TPICK_LAY_VENTOSE;		(* valorizzo la tipologia di prelievo = tipo prelievo falda *)
	END_IF
	
	Mission^.XPick			:= WorkArea^[Mission^.PPick].X;// + (Layer^[WorkArea^[Mission^.PPick].Layer].X / 2); (* valorizzo la quota X di prelievo  *)
	Mission^.YPick			:= WorkArea^[Mission^.PPick].Y + (Layer^[WorkPickPointState^[Mission^.PPick].Code].YDim / 2); (* valorizzo la quota Y di prelievo *)
	Mission^.ZPick			:= WorkArea^[Mission^.PPick].Z; (* in questo modo LA LENTA va sempre fino a zero...mi fermo al raggiungimento dell'intervento dei tastatori *)
ELSE
	Errore.Code := ErrWAM_TipologiaMagazzinoFaldaNONRiconosciuta; (*Errore, Nell'impianto è stata impostata una tipologia di magazzino falde non prevista!!!*)
	RETURN;//EXIT;
END_IF
//IF WorkAreaState^[cwa].P = 0 THEN (* Se devo depositare la falda su una CASSA/CAVALLETTO *)
//(*******************************************************************************************************************************)	
//(********************************************* DEPOSITO FALDA SU CASSA/CAVALLETTO **********************************************)
//(*******************************************************************************************************************************)
TFWAM_CreaMissione_DepFaldaSuPallet(NPosInLavoro			:= Mission^.PPlace, //Numero Postazione di depositio
									Angolo_Destinazione 	:= Forming^[WorkAreaState^[Mission^.PPlace].F].PElement[WorkAreaState^[Mission^.PPlace].P].J, //Angolo di deposito dell'elemento
									PosizioneAttuale_X      := ModuleAX_X^.Ax^.Status.ActPosition, //Posizione attuale asse X
									TipologiaTraiettoria    := Forming^[WorkAreaState^[cwa].F].PElement[WorkAreaState^[cwa].P].Trajectory,
									
									Quota_PostX				:= WorkArea^[Mission^.PPlace].X, //Quota X Postazione
									Quota_PostY				:= WorkArea^[Mission^.PPlace].Y, //Quota Y Postazione
									Quota_PostZ				:= WorkArea^[Mission^.PPlace].Z, //Quota Z Postazione
									Quota_PostJ				:= WorkArea^[Mission^.PPlace].Rx, //Quota J Postazione
									
									Offset_Postazione_X 	:= WorkAreaOffset^[Mission^.PPlace].X, //Offset X Postazione
									Offset_Postazione_Y 	:= WorkAreaOffset^[Mission^.PPlace].Y, //Offset Y Postazione
									Offset_Postazione_Z 	:= WorkAreaOffset^[Mission^.PPlace].Z, //Offset Z Postazione
									Offset_Postazione_J 	:= WorkAreaOffset^[Mission^.PPlace].Rx, //Offset J Postazione
									
									Pallet_DimX				:= Forming^[WorkAreaState^[Mission^.PPlace].F].Pallet.XDim, //Dimensione X Pallet
									Pallet_DimY				:= Forming^[WorkAreaState^[Mission^.PPlace].F].Pallet.YDim, //Dimensione Y Pallet
									Pallet_DimZ				:= Forming^[WorkAreaState^[Mission^.PPlace].F].Pallet.ZDim, //Dimensione Z Pallet
									
									Offset_Pallet_X_0		:= Forming^[WorkAreaState^[Mission^.PPlace].F].Pallet.OFSDE_X0, //Offset X Pallet o Casse
									Offset_Pallet_Y_0		:= Forming^[WorkAreaState^[Mission^.PPlace].F].Pallet.OFSDE_Y0, //Offset Y Pallet o Casse 
									Offset_Pallet_Z_0		:= Forming^[WorkAreaState^[Mission^.PPlace].F].Pallet.OFSDE_Z0, //Offset Z Pallet o Casse + è grande + il deposito si distanzia dal supporto
									Offset_Pallet_J_0		:= Forming^[WorkAreaState^[Mission^.PPlace].F].Pallet.OFSDE_J0, //Offset J Pallet o Casse + è grande + la lastra sarà inclinata verso l'angolo crescente
									
									Offset_Pallet_X_90		:= Forming^[WorkAreaState^[Mission^.PPlace].F].Pallet.OFSDE_X90, //Offset X Pallet lato 0-90 
									Offset_Pallet_Y_90		:= Forming^[WorkAreaState^[Mission^.PPlace].F].Pallet.OFSDE_Y90, //Offset Y Pallet lato 0-90 + è grande + il deposito si distanzia dal supporto
									Offset_Pallet_Z_90		:= Forming^[WorkAreaState^[Mission^.PPlace].F].Pallet.OFSDE_Z90, //Offset Z Pallet lato 0-90 + è grande + il deposito si distanzia dal supporto
									Offset_Pallet_J_90		:= Forming^[WorkAreaState^[Mission^.PPlace].F].Pallet.OFSDE_J90, //Offset J Pallet lato 0-90 + è grande + la lastra sarà inclinata in fase di deposito
									
									Offset_Pallet_X_180		:= Forming^[WorkAreaState^[Mission^.PPlace].F].Pallet.OFSDE_X180, //Offset X Pallet lato 90-180
									Offset_Pallet_Y_180		:= Forming^[WorkAreaState^[Mission^.PPlace].F].Pallet.OFSDE_Y180, //Offset Y Pallet lato 90-180 + è grande + il deposito si distanzia dal supporto
									Offset_Pallet_Z_180		:= Forming^[WorkAreaState^[Mission^.PPlace].F].Pallet.OFSDE_Z180, //Offset Z Pallet lato 90-180 + è grande + il deposito si distanzia dal supporto
									Offset_Pallet_J_180		:= Forming^[WorkAreaState^[Mission^.PPlace].F].Pallet.OFSDE_J180, //Offset J Pallet lato 90-180 + è grande + la lastra sarà inclinata in fase di deposito
									
									Quota_FormaturaX 		:= Forming^[WorkAreaState^[Mission^.PPlace].F].PElement[WorkAreaState^[Mission^.PPlace].P].X, //Quota Deposito X da Formatura
									Quota_FormaturaY 		:= Forming^[WorkAreaState^[Mission^.PPlace].F].PElement[WorkAreaState^[Mission^.PPlace].P].Y, //Quota Deposito Y da Formatura
									Quota_FormaturaZ 		:= Forming^[WorkAreaState^[Mission^.PPlace].F].PElement[WorkAreaState^[Mission^.PPlace].P].Z, //Quota Deposito Z da Formatura
									Quota_FormaturaJ 		:= Forming^[WorkAreaState^[Mission^.PPlace].F].PElement[WorkAreaState^[Mission^.PPlace].P].J, //Quota Deposito Z da Formatura
									
									Distanza_ApproccioFormaturaX 		:= Forming^[WorkAreaState^[Mission^.PPlace].F].PElement[WorkAreaState^[Mission^.PPlace].P].AX, //Distanza Deposito X da Formatura
									Distanza_ApproccioFormaturaY 		:= Forming^[WorkAreaState^[Mission^.PPlace].F].PElement[WorkAreaState^[Mission^.PPlace].P].AY, //Distanza Deposito Y da Formatura
									Distanza_ApproccioFormaturaZ 		:= Forming^[WorkAreaState^[Mission^.PPlace].F].PElement[WorkAreaState^[Mission^.PPlace].P].AZ, //Distanza Deposito Z da Formatura
									Distanza_ApproccioFormaturaJ 		:= Forming^[WorkAreaState^[Mission^.PPlace].F].PElement[WorkAreaState^[Mission^.PPlace].P].AJ, //Distanza Deposito Z da Formatura
									
									Quota_DestX 			=> Mission^.XPlace, //Quota DESTINAZIONE X
									Quota_DestY 			=> Mission^.YPlace, //Quota DESTINAZIONE Y
									Quota_DestZ 			=> Mission^.ZPlace, //Quota DESTINAZIONE Z
									Quota_DestJ 			=> Mission^.JPlace, //Quota DESTINAZIONE J	
									
									Quota_ApproccioDestX 	=> Mission^.XPlaceApproach, //Quota APPROCCIO di DESTINAZIONE X
									Quota_ApproccioDestY 	=> Mission^.YPlaceApproach, //Quota APPROCCIO di DESTINAZIONE Y
									Quota_ApproccioDestZ 	=> Mission^.ZPlaceApproach, //Quota APPROCCIO di DESTINAZIONE Z
									Quota_ApproccioDestJ 	=> Mission^.JPlaceApproach);//Quota APPROCCIO di DESTINAZIONE J	
	IF TFWAM_CreaMissione_DepFaldaSuPallet.Errore.Code > 0 THEN
		Errore := TFWAM_CreaMissione_DepFaldaSuPallet.Errore;
		RETURN;//EXIT;
	END_IF
	CASE Forming^[WorkAreaState^[Mission^.PPlace].F].Pallet.Tipologia OF
		CAVALLETTO :
			IF Forming^[WorkAreaState^[Mission^.PPlace].F].PElement[WorkAreaState^[Mission^.PPlace].P].J > 90 THEN (* Se devo depositare la falda su CAVALLETTO lato 180°*)	
				Mission^.XDim			:= Layer^[Forming^[WorkAreaState^[cwa].F].PElement[WorkAreaState^[Mission^.PPlace].P].TypologyCode].XDim ;
				Mission^.YDim			:= Layer^[Forming^[WorkAreaState^[cwa].F].PElement[WorkAreaState^[Mission^.PPlace].P].TypologyCode].YDim;
				Mission^.ZDim			:= Layer^[Forming^[WorkAreaState^[cwa].F].PElement[WorkAreaState^[Mission^.PPlace].P].TypologyCode].ZDim;
			ELSIF Forming^[WorkAreaState^[Mission^.PPlace].F].PElement[WorkAreaState^[Mission^.PPlace].P].J < 90 THEN (* Se devo depositare la falda su CAVALLETTO lato 0°*)		
				Mission^.XDim			:= Layer^[Forming^[WorkAreaState^[cwa].F].PElement[WorkAreaState^[Mission^.PPlace].P].TypologyCode].XDim ;
				Mission^.YDim			:= Layer^[Forming^[WorkAreaState^[cwa].F].PElement[WorkAreaState^[Mission^.PPlace].P].TypologyCode].YDim;
				Mission^.ZDim			:= Layer^[Forming^[WorkAreaState^[cwa].F].PElement[WorkAreaState^[Mission^.PPlace].P].TypologyCode].ZDim;
			END_IF
			WorkAreaManager^.State := WAMANAGER_CICLO_PRELIEVO_FALDA_RUN;	(* Set Stato del WorkAreaManager *)
			RestoreCWA^ := TRUE;
			PreviousPWA^ := pwa;
			RETURN;//EXIT;
		CASSA_STANDARD :
			Mission^.XDim			:= Layer^[Forming^[WorkAreaState^[cwa].F].PElement[WorkAreaState^[Mission^.PPlace].P].TypologyCode].XDim ;
			Mission^.YDim			:= Layer^[Forming^[WorkAreaState^[cwa].F].PElement[WorkAreaState^[Mission^.PPlace].P].TypologyCode].YDim;
			Mission^.ZDim			:= Layer^[Forming^[WorkAreaState^[cwa].F].PElement[WorkAreaState^[Mission^.PPlace].P].TypologyCode].ZDim;
			WorkAreaManager^.State := WAMANAGER_CICLO_PRELIEVO_FALDA_RUN;	(* Set Stato del WorkAreaManager *)
			RestoreCWA^ := TRUE;
			PreviousPWA^ := pwa;
			RETURN;//EXIT;
	ELSE
		Errore.Code := ErrWAM_TipologiaPalletNONRiconosciuta; 		(* Genero un errore che mi indica che la tipologia di "Pallet/Cassa/Cavallina" non è riconosciuto *)
		RETURN;//EXIT;		
	END_CASE
END_ACTION

ACTION LASTRA_PP_INIT:
(* Reset della memoria utilizzata per forzare il ciclo di riposo in ciclo di prelievo pacco *)
ForzaPrelievoPaccoDuranteCicloDiRiposo := FALSE;			
(* Definisco che la WORKAREA è positiva -> Default per lastre! *)
Mission^.PPick 	:= ppick;								   			// Assegno il numero del Punto di prelievo
Mission^.TPick 	:= TPICK_LASTRA;									// Assegno il tipo di Prelievo
Mission^.PPlace := cwa;									   			// Assegno il numero della piazzola di deposito
Mission^.XDim 	:= WorkPickPointState^[Mission^.PPick].Element.XDim ; 	// Assegno la dimensione X del pacco presente nel punto di prelievo designato
Mission^.YDim 	:= WorkPickPointState^[Mission^.PPick].Element.YDim; 	// Assegno la dimensione X del pacco presente nel punto di prelievo designato
Mission^.ZDim 	:= WorkPickPointState^[Mission^.PPick].Element.ZDim; 	// Assegno la dimensione X del pacco presente nel punto di prelievo designato

(* Calcolo Delle quote di Prelievo *)
XPick := TFPalletizer_CalcolaCoordinataPrelievo_PickPoint(WorkPickPoint,WorkPickPointState,WorkPickPointOffset,Mission^.PPick,'X');		
YPick := TFPalletizer_CalcolaCoordinataPrelievo_PickPoint(WorkPickPoint,WorkPickPointState,WorkPickPointOffset,Mission^.PPick,'Y');
ZPick := TFPalletizer_CalcolaCoordinataPrelievo_PickPoint(WorkPickPoint,WorkPickPointState,WorkPickPointOffset,Mission^.PPick,'Z');
JPick := TFPalletizer_CalcolaCoordinataPrelievo_PickPoint(WorkPickPoint,WorkPickPointState,WorkPickPointOffset,Mission^.PPick,'J');	

(* Assegnazione quote alla Missione *)
Mission^.XPick			:= XPick;
Mission^.YPick			:= YPick;
Mission^.ZPick			:= ZPick;
Mission^.JPick			:= JPick;

Mission^.XPickApproach	:= XPick;							
Mission^.YPickApproach	:= YPick;	  
Mission^.ZPickApproach	:= ZPick + PickPlaceParameters^.ZPickApproach;//Quota prelievo + offset approccio... in mod da fare la lenta ottimizzata
Mission^.JPickApproach	:= JPick;	
	
(* Set delle variabili per andare al punto di riposo *)
X_Riposo	:= XPick;
Y_Riposo	:= YPick;
J_Riposo	:= JPick;
Z_Riposo	:= QuotaFuoriIngombro_Z_AVUOTO;		

IF WorkAreaState^[Mission^.PPlace].Apprendimento.Z.Lato90.Stato <> APPRENDIMENTO_ESEGUITO THEN
	IF WorkareaState^[Mission^.PPlace].TransportState.Supporto.Tipologia = e_Tipo_Pallet.CASSA_STANDARD THEN 
		WorkAreaState^[Mission^.PPlace].Apprendimento.Z.Lato90.QuotaStart 	:= 950;
	ELSE
		WorkAreaState^[Mission^.PPlace].Apprendimento.Z.Lato90.QuotaStart 	:= 950;
	END_IF
END_IF
//Disabilito apprendimento in deposito se disabilitato
IF NOT HMI_AbilitaDepositoPaccoOrrizzontaleConTasteggio THEN
	WorkAreaState^[Mission^.PPlace].Apprendimento.Z.Lato90.Stato := APPRENDIMENTO_DISABILITATO;
END_IF
(* Calcolo gli ingombri della pinza nelle varie direzioni *)
IF Forming^[WorkAreaState^[Mission^.PPlace].F].PElement[WorkAreaState^[Mission^.PPlace].P].J <= 87 THEN
	LatoDeposito := 0;
ELSIF Forming^[WorkAreaState^[Mission^.PPlace].F].PElement[WorkAreaState^[Mission^.PPlace].P].J >= 93 THEN
	LatoDeposito := 180;
END_IF
							
TFCalcoliIngombroPinza(Mission := Mission,
					WorkAreaManager := WorkAreaManager,
					WorkAreaState := ADR(WorkAreaState),
					ModuleAX_J := ModuleAX_J,
					AngoloRotazioneDestinazionePinza:= Forming^[WorkAreaState^[Mission^.PPlace].F].PElement[WorkAreaState^[Mission^.PPlace].P].J,
					IngombroX_Pos 				:= ADR(IngombroX_Pos),
					IngombroY_Pos 				:= ADR(IngombroY_Pos),
					IngombroX_Neg 				:= ADR(IngombroX_Neg),
					IngombroY_Neg 				:= ADR(IngombroY_Neg),
					IngombroZ_Pos 				:= ADR(IngombroZ_Pos),
					IngombroZ_Neg 				:= ADR(IngombroZ_Neg),
					IngombroY_Tot 				:= ADR(IngombroY_Tot),
					IngombroDestinazioneX_Pos 	:= ADR(IngombroDestinazioneX_Pos),
					IngombroDestinazioneY_Pos 	:= ADR(IngombroDestinazioneY_Pos),
					IngombroDestinazioneX_Neg 	:= ADR(IngombroDestinazioneX_Neg),
					IngombroDestinazioneY_Neg 	:= ADR(IngombroDestinazioneY_Neg),
					IngombroDestinazioneZ_Pos 	:= ADR(IngombroDestinazioneZ_Pos),
					IngombroDestinazioneZ_Neg 	:= ADR(IngombroDestinazioneZ_Neg),
					IngombroMaxX_Pos 			:= ADR(IngombroMaxX_Pos),
					IngombroMaxY_Pos 			:= ADR(IngombroMaxY_Pos),
					IngombroMaxX_Neg 			:= ADR(IngombroMaxX_Neg),
					IngombroMaxY_Neg 			:= ADR(IngombroMaxY_Neg),
					IngombroMaxZ_Pos 			:= ADR(IngombroMaxZ_Pos),
					IngombroMaxZ_Neg 			:= ADR(IngombroMaxZ_Neg),
					IngombroY_Pos_0  			:= ADR(IngombroY_Pos_0),		 		
					IngombroY_Neg_180 			:= ADR(IngombroY_Neg_180),
					IngombroY_Neg_0 			:= ADR(IngombroY_Neg_0),	
					IngombroY_Pos_180 			:= ADR(IngombroY_Pos_180),
					ScostamentoVerticalePuntoCentrale := ADR(ScostamentoVerticalePuntoCentrale));

(* Valorizzazione quote di deposito Ciclo Lastra *)
TFWAM_CreaMissione_DepLastraDaPP(NPosInLavoro			    := Mission^.PPlace, //Numero Postazione di depositio
									Angolo_Destinazione 	:= Forming^[WorkAreaState^[Mission^.PPlace].F].PElement[WorkAreaState^[Mission^.PPlace].P].J, //Angolo di deposito dell'elemento
									PosizioneAttuale_X      := ModuleAX_X^.Ax^.Status.ActPosition, //Posizione attuale asse X
									TipologiaTraiettoria    := TRAIETTORIA_CON_APPROCCIO,//Forming^[WorkAreaState^[cwa].F].PElement[WorkAreaState^[cwa].P].Trajectory,
									Apprendimento			:= WorkAreaState^[Mission^.PPlace].Apprendimento,
									CicloDiPrelievo         := FALSE,
									HmaxElemento			:= WorkAreaState^[Mission^.PPlace].TransportState.Supporto.HMAX,
									Offset_Apprendimento_X 	:= 0,//OffsetApprendimento.Lastra.X, //Offset X Postazione,
									Offset_Apprendimento_Y 	:= OffsetApprendimento.Lastra.Y, //Offset Y Postazione
									Offset_Apprendimento_Z 	:= OffsetApprendimento.Lastra.Z, //Offset Z Postazione
									Offset_Apprendimento_J 	:= 0,//OffsetApprendimento.Lastra.J, //Offset J Postazione

									Quota_PostX				:= WorkArea^[Mission^.PPlace].X, //Quota X Postazione
									Quota_PostY				:= WorkArea^[Mission^.PPlace].Y, //Quota Y Postazione
									Quota_PostZ				:= WorkArea^[Mission^.PPlace].Z, //Quota Z Postazione
									Quota_PostJ				:= WorkArea^[Mission^.PPlace].Rx, //Quota J Postazione
									
									Offset_Postazione_X 	:= WorkAreaOffset^[Mission^.PPlace].X, //Offset X Postazione
									Offset_Postazione_Y 	:= WorkAreaOffset^[Mission^.PPlace].Y, //Offset Y Postazione
									Offset_Postazione_Z 	:= WorkAreaOffset^[Mission^.PPlace].Z, //Offset Z Postazione
									Offset_Postazione_J 	:= WorkAreaOffset^[Mission^.PPlace].Rx, //Offset J Postazione
									
									Pallet_DimX				:= WorkAreaState^[Mission^.PPlace].Supporto.XDim, //Dimensione X Pallet
									Pallet_DimY				:= WorkAreaState^[Mission^.PPlace].Supporto.YDim, //Dimensione Y Pallet
									Pallet_DimZ				:= WorkAreaState^[Mission^.PPlace].Supporto.ZDim, //Dimensione Z Pallet
									
									Quota_FormaturaX 		:= Forming^[WorkAreaState^[Mission^.PPlace].F].PElement[WorkAreaState^[Mission^.PPlace].P].X, //Quota Deposito X da Formatura
									Quota_FormaturaY 		:= ABS(Forming^[WorkAreaState^[Mission^.PPlace].F].PElement[WorkAreaState^[Mission^.PPlace].P].Y), //Quota Deposito Y da Formatura
									Quota_FormaturaZ 		:= Forming^[WorkAreaState^[Mission^.PPlace].F].PElement[WorkAreaState^[Mission^.PPlace].P].Z, //Quota Deposito Z da Formatura
									Quota_FormaturaJ 		:= Forming^[WorkAreaState^[Mission^.PPlace].F].PElement[WorkAreaState^[Mission^.PPlace].P].J, //Quota Deposito Z da Formatura
									
									Distanza_ApproccioFormaturaX 		:= Forming^[WorkAreaState^[Mission^.PPlace].F].PElement[WorkAreaState^[Mission^.PPlace].P].AX, //Quota Deposito X da Formatura
									Distanza_ApproccioFormaturaY 		:= PickPlaceParameters^.YPlaceApproach, 
									Distanza_ApproccioFormaturaZ 		:= PickPlaceParameters^.ZPlaceApproach,
									Distanza_ApproccioFormaturaJ 		:= Forming^[WorkAreaState^[Mission^.PPlace].F].PElement[WorkAreaState^[Mission^.PPlace].P].AJ, //Quota Deposito Z da Formatura
									
									Quota_DestX 			=> Mission^.XPlace, //Quota DESTINAZIONE X
									Quota_DestY 			=> Mission^.YPlace, //Quota DESTINAZIONE Y
									Quota_DestZ 			=> Mission^.ZPlace, //Quota DESTINAZIONE Z
									Quota_DestJ 			=> Mission^.JPlace, //Quota DESTINAZIONE J	
									
									Quota_ApproccioDestX 	=> Mission^.XPlaceApproach, //Quota APPROCCIO di DESTINAZIONE X
									Quota_ApproccioDestY 	=> Mission^.YPlaceApproach, //Quota APPROCCIO di DESTINAZIONE Y
									Quota_ApproccioDestZ 	=> Mission^.ZPlaceApproach, //Quota APPROCCIO di DESTINAZIONE Z
									Quota_ApproccioDestJ 	=> Mission^.JPlaceApproach);//Quota APPROCCIO di DESTINAZIONE J	

IF TFWAM_CreaMissione_DepLastraDaPP.Errore.Code > 0 THEN
	Errore := TFWAM_CreaMissione_DepLastraDaPP.Errore;
	RETURN;//EXIT;
ELSE
	RestoreCWA^ := TRUE;
	PreviousPWA^ := pwa;
	WorkAreaManager^.State 	:= WAMANAGER_CICLO_PRELIEVO_LASTRA_PP_RUN;
END_IF
(* Setto l'uscita che mi determina il deposito del primo pacco in lenta *)
IF WorkAreaState^[Mission^.PPlace].Slow = 1 THEN
	DepositoPaccoInLenta := TRUE;
END_IF
END_ACTION

